C07276=1022.526,-49.278,404.640,166.557,49.308,158.966
C07277=1022.532,-49.029,404.628,166.560,49.304,158.966
C07278=1022.538,-48.778,404.616,166.563,49.300,158.966
C07279=1022.544,-48.529,404.605,166.566,49.296,158.965
C07280=1022.550,-48.279,404.592,166.568,49.292,158.965
C07281=1022.555,-48.030,404.581,166.572,49.289,158.965
C07282=1022.561,-47.780,404.569,166.574,49.285,158.965
C07283=1022.566,-47.530,404.557,166.577,49.281,158.964
C07284=1022.573,-47.281,404.545,166.580,49.277,158.964
C07285=1022.578,-47.031,404.534,166.583,49.274,158.964
C07286=1022.585,-46.781,404.522,166.586,49.270,158.964
C07287=1022.590,-46.532,404.510,166.588,49.266,158.963
C07288=1022.596,-46.282,404.498,166.592,49.263,158.963
C07289=1022.601,-46.033,404.486,166.594,49.259,158.963
C07290=1022.607,-45.783,404.474,166.598,49.254,158.963
C07291=1022.613,-45.533,404.463,166.601,49.251,158.963
C07292=1022.619,-45.284,404.450,166.604,49.247,158.962
C07293=1022.625,-45.035,404.439,166.607,49.243,158.962
C07294=1022.631,-44.784,404.427,166.610,49.239,158.962
C07295=1022.636,-44.535,404.415,166.613,49.236,158.962
C07296=1022.643,-44.285,404.403,166.615,49.232,158.961
C07297=1022.648,-44.035,404.391,166.618,49.228,158.961
C07298=1022.654,-43.786,404.379,166.621,49.224,158.961
C07299=1022.660,-43.536,404.367,166.624,49.221,158.961
C07300=1022.666,-43.287,404.356,166.627,49.217,158.960
C07301=1022.672,-43.037,404.343,166.630,49.213,158.960
C07302=1022.677,-42.788,404.331,166.632,49.209,158.960
C07303=1022.684,-42.538,404.319,166.635,49.205,158.960
C07304=1022.689,-42.288,404.307,166.638,49.201,158.959
C07305=1022.695,-42.039,404.296,166.642,49.197,158.959
C07306=1022.701,-41.789,404.283,166.645,49.193,158.959
C07307=1022.707,-41.539,404.271,166.648,49.189,158.958
C07308=1022.713,-41.289,404.260,166.651,49.186,158.958
C07309=1022.719,-41.040,404.247,166.653,49.182,158.958
C07310=1022.725,-40.791,404.236,166.656,49.178,158.958
C07311=1022.731,-40.541,404.223,166.659,49.174,158.957
C07312=1022.737,-40.291,404.210,166.662,49.170,158.957
C07313=1022.743,-40.041,404.200,166.665,49.167,158.957
C07314=1022.748,-39.792,404.187,166.668,49.163,158.957
C07315=1022.755,-39.542,404.175,166.670,49.159,158.956
C07316=1022.760,-39.293,404.163,166.673,49.155,158.956
C07317=1022.766,-39.043,404.150,166.676,49.151,158.956
C07318=1022.772,-38.793,404.138,166.679,49.147,158.956
C07319=1022.779,-38.543,404.126,166.682,49.143,158.955
C07320=1022.784,-38.294,404.114,166.685,49.139,158.955
C07321=1022.790,-38.044,404.101,166.688,49.136,158.955
C07322=1022.796,-37.794,404.089,166.690,49.132,158.955
C07323=1022.801,-37.545,404.077,166.693,49.128,158.954
C07324=1022.808,-37.266,404.063,166.697,49.124,158.954
C07325=1022.815,-36.986,404.049,166.700,49.120,158.954
C07326=1022.821,-36.708,404.035,166.704,49.116,158.954
C07327=1022.828,-36.429,404.021,166.706,49.112,158.953
C07328=1022.834,-36.179,404.008,166.709,49.108,158.953
C07329=1022.839,-35.929,403.996,166.712,49.104,158.953
C07330=1022.845,-35.680,403.984,166.715,49.100,158.953
C07331=1022.851,-35.430,403.972,166.718,49.096,158.952
C07332=1022.857,-35.180,403.959,166.721,49.093,158.952
C07333=1022.863,-34.931,403.947,166.724,49.089,158.952
C07334=1022.869,-34.681,403.934,166.726,49.085,158.952
C07335=1022.875,-34.431,403.922,166.729,49.081,158.951
C07336=1022.880,-34.181,403.909,166.732,49.078,158.951
C07337=1022.886,-33.932,403.897,166.735,49.074,158.951
C07338=1022.892,-33.682,403.885,166.738,49.070,158.951
C07339=1022.898,-33.433,403.873,166.741,49.066,158.950
C07340=1022.904,-33.183,403.859,166.744,49.063,158.950
C07341=1022.910,-32.934,403.847,166.747,49.059,158.950
C07342=1022.916,-32.684,403.835,166.749,49.055,158.950
C07343=1022.922,-32.434,403.822,166.752,49.051,158.949
C07344=1022.928,-32.185,403.809,166.755,49.048,158.949
C07345=1022.933,-31.935,403.797,166.758,49.044,158.949
C07346=1022.939,-31.686,403.785,166.761,49.040,158.949
C07347=1022.945,-31.436,403.771,166.764,49.036,158.948
C07348=1022.952,-31.187,403.760,166.767,49.032,158.948
C07349=1022.958,-30.937,403.747,166.769,49.028,158.948
C07350=1022.963,-30.687,403.734,166.772,49.024,158.948
C07351=1022.969,-30.437,403.722,166.775,49.020,158.947
C07352=1022.975,-30.188,403.709,166.778,49.017,158.947
C07353=1022.981,-29.939,403.696,166.781,49.013,158.947
C07354=1022.987,-29.689,403.684,166.784,49.009,158.946
C07355=1022.993,-29.439,403.671,166.786,49.005,158.946
C07356=1022.999,-29.189,403.659,166.789,49.001,158.946
C07357=1023.006,-28.940,403.646,166.792,48.997,158.946
C07358=1023.011,-28.690,403.634,166.795,48.994,158.945
C07359=1023.017,-28.441,403.621,166.798,48.990,158.945
C07360=1023.023,-28.192,403.608,166.801,48.986,158.945
C07361=1023.029,-27.942,403.595,166.804,48.982,158.945
C07362=1023.035,-27.692,403.583,166.807,48.978,158.944
C07363=1023.041,-27.442,403.570,166.810,48.974,158.944
C07364=1023.047,-27.193,403.557,166.812,48.971,158.944
C07365=1023.053,-26.943,403.545,166.815,48.967,158.943
C07366=1023.059,-26.694,403.531,166.818,48.963,158.943
C07367=1023.064,-26.443,403.518,166.821,48.960,158.943
C07368=1023.070,-26.194,403.506,166.824,48.956,158.943
C07369=1023.076,-25.945,403.493,166.826,48.952,158.942
C07370=1023.082,-25.695,403.480,166.829,48.949,158.942
C07371=1023.088,-25.446,403.467,166.832,48.945,158.942
C07372=1023.094,-25.196,403.454,166.835,48.941,158.942
C07373=1023.099,-24.946,403.440,166.838,48.938,158.942
C07374=1023.105,-24.696,403.428,166.841,48.934,158.941
C07375=1023.111,-24.447,403.415,166.844,48.930,158.941
C07376=1023.117,-24.197,403.402,166.847,48.926,158.941
C07377=1023.123,-23.948,403.389,166.850,48.922,158.941
C07378=1023.129,-23.698,403.376,166.852,48.918,158.940
C07379=1023.135,-23.449,403.362,166.854,48.915,158.940
C07380=1023.141,-23.199,403.350,166.857,48.912,158.940
C07381=1023.147,-22.949,403.337,166.860,48.908,158.939
C07382=1023.153,-22.700,403.324,166.863,48.904,158.939
C07383=1023.159,-22.450,403.311,166.866,48.900,158.939
C07384=1023.164,-22.200,403.298,166.869,48.896,158.939
C07385=1023.170,-21.951,403.284,166.871,48.892,158.938
C07386=1023.176,-21.701,403.272,166.874,48.889,158.938
C07387=1023.183,-21.452,403.258,166.877,48.885,158.938
C07388=1023.189,-21.172,403.244,166.880,48.881,158.937
C07389=1023.196,-20.892,403.229,166.884,48.876,158.937
C07390=1023.202,-20.612,403.214,166.886,48.872,158.937
C07391=1023.209,-20.332,403.200,166.890,48.867,158.937
C07392=1023.215,-20.083,403.187,166.893,48.864,158.936
C07393=1023.221,-19.833,403.174,166.896,48.860,158.936
C07394=1023.227,-19.582,403.160,166.899,48.856,158.936
C07395=1023.233,-19.333,403.147,166.901,48.852,158.935
C07396=1023.239,-19.084,403.134,166.903,48.849,158.935
C07397=1023.245,-18.834,403.121,166.906,48.845,158.935
C07398=1023.251,-18.585,403.108,166.909,48.842,158.935
C07399=1023.257,-18.335,403.094,166.912,48.838,158.934
C07400=1023.263,-18.085,403.081,166.915,48.834,158.934
C07401=1023.269,-17.836,403.068,166.917,48.830,158.934
C07402=1023.275,-17.587,403.055,166.921,48.826,158.934
C07403=1023.281,-17.337,403.042,166.923,48.822,158.933
C07404=1023.287,-17.087,403.028,166.926,48.819,158.933
C07405=1023.293,-16.838,403.015,166.929,48.815,158.933
C07406=1023.299,-16.588,403.003,166.932,48.811,158.932
C07407=1023.305,-16.339,402.989,166.934,48.807,158.932
C07408=1023.312,-16.089,402.976,166.938,48.803,158.932
C07409=1023.317,-15.839,402.962,166.940,48.800,158.932
C07410=1023.323,-15.589,402.949,166.943,48.796,158.931
C07411=1023.329,-15.340,402.936,166.946,48.792,158.931
C07412=1023.335,-15.091,402.922,166.949,48.788,158.931
C07413=1023.341,-14.841,402.909,166.951,48.785,158.930
C07414=1023.346,-14.592,402.895,166.954,48.781,158.930
C07415=1023.353,-14.343,402.882,166.956,48.777,158.930
C07416=1023.359,-14.092,402.868,166.960,48.774,158.930
C07417=1023.365,-13.842,402.855,166.962,48.770,158.929
C07418=1023.370,-13.593,402.841,166.965,48.766,158.929
C07419=1023.376,-13.344,402.828,166.968,48.763,158.929
C07420=1023.382,-13.094,402.814,166.971,48.759,158.929
C07421=1023.388,-12.845,402.801,166.973,48.755,158.928
C07422=1023.394,-12.595,402.787,166.976,48.751,158.928
C07423=1023.400,-12.345,402.773,166.979,48.748,158.928
C07424=1023.406,-12.096,402.759,166.982,48.744,158.927
C07425=1023.412,-11.846,402.746,166.984,48.740,158.927
C07426=1023.418,-11.597,402.732,166.987,48.736,158.927
C07427=1023.424,-11.347,402.719,166.990,48.733,158.927
C07428=1023.429,-11.098,402.705,166.993,48.729,158.926
C07429=1023.436,-10.848,402.691,166.996,48.725,158.926
C07430=1023.442,-10.598,402.678,166.998,48.721,158.926
C07431=1023.448,-10.349,402.664,167.001,48.718,158.925
C07432=1023.454,-10.100,402.651,167.004,48.714,158.925
C07433=1023.459,-9.850,402.637,167.006,48.710,158.925
C07434=1023.466,-9.600,402.624,167.009,48.706,158.924
C07435=1023.472,-9.351,402.610,167.012,48.703,158.924
C07436=1023.478,-9.101,402.596,167.015,48.699,158.924
C07437=1023.483,-8.852,402.583,167.018,48.695,158.924
C07438=1023.490,-8.602,402.569,167.021,48.691,158.923
C07439=1023.496,-8.352,402.555,167.022,48.687,158.923
C07440=1023.502,-8.103,402.542,167.025,48.684,158.923
C07441=1023.507,-7.854,402.528,167.028,48.680,158.923
C07442=1023.514,-7.604,402.515,167.031,48.676,158.922
C07443=1023.520,-7.354,402.500,167.034,48.672,158.922
C07444=1023.526,-7.105,402.487,167.037,48.669,158.922
C07445=1023.531,-6.855,402.473,167.039,48.665,158.921
C07446=1023.538,-6.605,402.460,167.042,48.661,158.921
C07447=1023.544,-6.356,402.445,167.045,48.657,158.921
C07448=1023.550,-6.107,402.432,167.047,48.654,158.920
C07449=1023.556,-5.857,402.418,167.050,48.650,158.920
C07450=1023.562,-5.607,402.404,167.053,48.646,158.920
C07451=1023.568,-5.358,402.390,167.056,48.642,158.919
C07452=1023.575,-5.076,402.375,167.059,48.638,158.919
C07453=1023.582,-4.794,402.359,167.062,48.633,158.919
C07454=1023.589,-4.513,402.344,167.065,48.629,158.918
C07455=1023.596,-4.231,402.329,167.069,48.625,158.918
C07456=1023.602,-3.981,402.314,167.071,48.621,158.918
C07457=1023.607,-3.732,402.300,167.073,48.618,158.917
C07458=1023.613,-3.483,402.286,167.076,48.614,158.917
C07459=1023.619,-3.232,402.272,167.079,48.610,158.917
C07460=1023.625,-2.983,402.258,167.082,48.606,158.917
C07461=1023.631,-2.734,402.244,167.085,48.603,158.917
C07462=1023.637,-2.484,402.230,167.087,48.600,158.916
C07463=1023.643,-2.234,402.216,167.090,48.596,158.916
C07464=1023.648,-1.985,402.201,167.093,48.592,158.916
C07465=1023.654,-1.735,402.187,167.095,48.589,158.915
C07466=1023.660,-1.486,402.172,167.098,48.585,158.915
C07467=1023.666,-1.236,402.158,167.100,48.582,158.915
C07468=1023.672,-0.986,402.144,167.103,48.578,158.915
C07469=1023.678,-0.738,402.130,167.106,48.574,158.914
C07470=1023.684,-0.488,402.116,167.109,48.570,158.914
C07471=1023.690,-0.238,402.101,167.112,48.567,158.914
C07472=1023.696,0.011,402.088,167.114,48.563,158.913
C07473=1023.701,0.261,402.074,167.116,48.559,158.913
C07474=1023.707,0.510,402.059,167.120,48.556,158.913
C07475=1023.713,0.760,402.045,167.122,48.552,158.913
C07476=1023.719,1.009,402.031,167.125,48.548,158.912
C07477=1023.726,1.259,402.017,167.127,48.545,158.912
C07478=1023.731,1.508,402.002,167.130,48.541,158.912
C07479=1023.737,1.758,401.988,167.133,48.537,158.911
C07480=1023.743,2.007,401.973,167.136,48.533,158.911
C07481=1023.749,2.257,401.959,167.139,48.530,158.911
C07482=1023.755,2.507,401.945,167.141,48.527,158.910
C07483=1023.761,2.756,401.931,167.143,48.523,158.910
C07484=1023.767,3.006,401.917,167.146,48.519,158.910
C07485=1023.773,3.255,401.902,167.149,48.515,158.909
C07486=1023.779,3.504,401.888,167.152,48.512,158.909
C07487=1023.785,3.754,401.874,167.154,48.508,158.909
C07488=1023.791,4.003,401.859,167.157,48.504,158.909
C07489=1023.797,4.253,401.845,167.160,48.500,158.908
C07490=1023.803,4.502,401.830,167.162,48.496,158.908
C07491=1023.809,4.753,401.816,167.166,48.493,158.908
C07492=1023.814,5.002,401.801,167.167,48.489,158.907
C07493=1023.821,5.251,401.788,167.170,48.486,158.907
C07494=1023.827,5.500,401.773,167.173,48.482,158.907
C07495=1023.833,5.751,401.759,167.176,48.478,158.906
C07496=1023.839,6.000,401.744,167.179,48.474,158.906
C07497=1023.845,6.249,401.729,167.182,48.471,158.906
C07498=1023.851,6.499,401.716,167.183,48.467,158.906
C07499=1023.857,6.749,401.701,167.186,48.463,158.905
C07500=1023.863,6.998,401.687,167.189,48.459,158.905
C07501=1023.869,7.248,401.672,167.192,48.455,158.905
C07502=1023.876,7.496,401.658,167.195,48.451,158.904
C07503=1023.882,7.747,401.644,167.197,48.449,158.904
C07504=1023.887,7.996,401.629,167.200,48.445,158.904
C07505=1023.894,8.245,401.614,167.202,48.441,158.903
C07506=1023.899,8.495,401.600,167.205,48.437,158.903
C07507=1023.906,8.745,401.585,167.208,48.433,158.903
C07508=1023.911,8.994,401.571,167.211,48.429,158.902
C07509=1023.918,9.244,401.556,167.213,48.425,158.902
C07510=1023.923,9.493,401.542,167.215,48.421,158.902
C07511=1023.930,9.742,401.527,167.218,48.418,158.901
C07512=1023.936,9.992,401.514,167.221,48.414,158.901
C07513=1023.942,10.241,401.499,167.224,48.410,158.901
C07514=1023.948,10.490,401.484,167.227,48.407,158.901
C07515=1023.954,10.740,401.469,167.229,48.403,158.900
C07516=1023.962,11.023,401.453,167.232,48.398,158.900
C07517=1023.968,11.307,401.436,167.235,48.394,158.899
C07518=1023.975,11.591,401.419,167.238,48.390,158.899
C07519=1023.982,11.874,401.403,167.242,48.385,158.899
C07520=1023.988,12.124,401.389,167.244,48.382,158.898
C07521=1023.994,12.373,401.374,167.247,48.378,158.898
C07522=1024.000,12.623,401.359,167.249,48.374,158.898
C07523=1024.007,12.873,401.344,167.252,48.370,158.897
C07524=1024.012,13.122,401.330,167.255,48.366,158.897
C07525=1024.019,13.372,401.316,167.257,48.362,158.897
C07526=1024.025,13.622,401.301,167.260,48.358,158.896
C07527=1024.031,13.871,401.286,167.262,48.356,158.896
C07528=1024.037,14.120,401.271,167.265,48.352,158.896
C07529=1024.043,14.369,401.257,167.268,48.348,158.895
C07530=1024.049,14.619,401.242,167.271,48.344,158.895
C07531=1024.055,14.869,401.226,167.273,48.340,158.895
C07532=1024.061,15.118,401.211,167.276,48.337,158.895
C07533=1024.067,15.367,401.197,167.278,48.333,158.894
C07534=1024.073,15.616,401.182,167.281,48.329,158.894
C07535=1024.079,15.866,401.167,167.284,48.325,158.894
C07536=1024.085,16.117,401.152,167.286,48.322,158.893
C07537=1024.090,16.366,401.138,167.289,48.319,158.893
C07538=1024.097,16.615,401.123,167.292,48.315,158.893
C07539=1024.103,16.865,401.108,167.295,48.311,158.892
C07540=1024.109,17.114,401.093,167.296,48.307,158.892
C07541=1024.115,17.364,401.078,167.299,48.303,158.892
C07542=1024.121,17.613,401.063,167.302,48.299,158.891
C07543=1024.127,17.862,401.048,167.305,48.296,158.891
C07544=1024.133,18.112,401.033,167.307,48.293,158.891
C07545=1024.139,18.362,401.018,167.310,48.289,158.890
C07546=1024.145,18.610,401.002,167.313,48.285,158.890
C07547=1024.151,18.860,400.987,167.316,48.281,158.890
C07548=1024.158,19.110,400.972,167.317,48.277,158.889
C07549=1024.163,19.359,400.958,167.320,48.274,158.889
C07550=1024.169,19.609,400.942,167.323,48.270,158.889
C07551=1024.175,19.858,400.927,167.326,48.266,158.888
C07552=1024.182,20.108,400.912,167.328,48.263,158.888
C07553=1024.187,20.357,400.897,167.331,48.259,158.888
C07554=1024.193,20.607,400.882,167.334,48.255,158.887
C07555=1024.200,20.857,400.867,167.336,48.251,158.887
C07556=1024.205,21.105,400.851,167.339,48.248,158.887
C07557=1024.211,21.355,400.836,167.341,48.244,158.886
C07558=1024.218,21.604,400.822,167.344,48.241,158.886
C07559=1024.223,21.854,400.806,167.347,48.237,158.886
C07560=1024.229,22.103,400.791,167.349,48.233,158.885
C07561=1024.235,22.353,400.776,167.352,48.229,158.885
C07562=1024.241,22.602,400.760,167.355,48.226,158.885
C07563=1024.247,22.851,400.746,167.358,48.222,158.885
C07564=1024.254,23.101,400.731,167.359,48.219,158.884
C07565=1024.259,23.351,400.715,167.362,48.215,158.884
C07566=1024.266,23.601,400.700,167.365,48.211,158.884
C07567=1024.272,23.850,400.684,167.368,48.207,158.883
C07568=1024.277,24.099,400.669,167.370,48.203,158.883
C07569=1024.284,24.349,400.654,167.373,48.200,158.883
C07570=1024.289,24.599,400.639,167.376,48.196,158.882
C07571=1024.296,24.848,400.623,167.378,48.192,158.882
C07572=1024.302,25.097,400.609,167.380,48.189,158.882
C07573=1024.308,25.347,400.593,167.383,48.185,158.881
C07574=1024.314,25.596,400.578,167.386,48.181,158.881
C07575=1024.321,25.845,400.562,167.389,48.177,158.881
C07576=1024.326,26.095,400.547,167.391,48.174,158.880
C07577=1024.332,26.344,400.532,167.394,48.170,158.880
C07578=1024.338,26.593,400.516,167.397,48.167,158.880
C07579=1024.344,26.843,400.501,167.398,48.163,158.879
C07580=1024.351,27.128,400.483,167.402,48.158,158.879
C07581=1024.358,27.413,400.466,167.405,48.154,158.878
C07582=1024.365,27.698,400.448,167.407,48.150,158.878
C07583=1024.372,27.983,400.430,167.411,48.146,158.878
C07584=1024.378,28.233,400.415,167.413,48.142,158.877
C07585=1024.384,28.482,400.399,167.416,48.138,158.877
C07586=1024.390,28.731,400.384,167.419,48.135,158.877
C07587=1024.396,28.981,400.369,167.421,48.131,158.876
C07588=1024.402,29.230,400.352,167.423,48.127,158.876
C07589=1024.408,29.480,400.337,167.426,48.124,158.876
C07590=1024.414,29.729,400.321,167.428,48.120,158.875
C07591=1024.420,29.978,400.307,167.431,48.117,158.875
C07592=1024.426,30.228,400.290,167.434,48.113,158.875
C07593=1024.431,30.478,400.275,167.436,48.109,158.874
C07594=1024.438,30.727,400.259,167.439,48.106,158.874
C07595=1024.444,30.977,400.244,167.442,48.102,158.874
C07596=1024.450,31.226,400.228,167.444,48.098,158.873
C07597=1024.456,31.476,400.212,167.447,48.095,158.873
C07598=1024.461,31.724,400.197,167.449,48.091,158.873
C07599=1024.468,31.974,400.182,167.452,48.087,158.872
C07600=1024.474,32.223,400.165,167.454,48.084,158.872
C07601=1024.480,32.473,400.150,167.457,48.080,158.872
C07602=1024.486,32.722,400.134,167.460,48.076,158.871
C07603=1024.492,32.972,400.118,167.462,48.072,158.871
C07604=1024.498,33.221,400.103,167.465,48.069,158.871
C07605=1024.504,33.471,400.087,167.467,48.065,158.870
C07606=1024.510,33.721,400.071,167.470,48.061,158.870
C07607=1024.516,33.969,400.056,167.472,48.058,158.870
C07608=1024.522,34.219,400.040,167.475,48.054,158.869
C07609=1024.528,34.468,400.025,167.478,48.050,158.869
C07610=1024.534,34.717,400.008,167.481,48.046,158.869
C07611=1024.540,34.967,399.993,167.482,48.043,158.868
C07612=1024.547,35.216,399.977,167.485,48.039,158.868
C07613=1024.552,35.466,399.962,167.488,48.035,158.868
C07614=1024.558,35.716,399.945,167.490,48.032,158.867
C07615=1024.565,35.965,399.930,167.493,48.028,158.867
C07616=1024.570,36.215,399.914,167.496,48.024,158.867
C07617=1024.577,36.464,399.899,167.499,48.021,158.866
C07618=1024.583,36.713,399.882,167.501,48.017,158.866
C07619=1024.589,36.963,399.867,167.503,48.013,158.866
C07620=1024.595,37.212,399.850,167.506,48.009,158.865
C07621=1024.601,37.462,399.834,167.508,48.006,158.865
C07622=1024.607,37.711,399.819,167.511,48.002,158.865
C07623=1024.613,37.961,399.803,167.514,47.999,158.864
C07624=1024.619,38.210,399.787,167.516,47.995,158.864
C07625=1024.625,38.460,399.770,167.519,47.991,158.864
C07626=1024.631,38.709,399.754,167.522,47.987,158.863
C07627=1024.637,38.958,399.738,167.523,47.984,158.863
C07628=1024.642,39.208,399.722,167.526,47.981,158.863
C07629=1024.649,39.457,399.707,167.529,47.977,158.862
C07630=1024.655,39.706,399.691,167.531,47.973,158.862
C07631=1024.660,39.955,399.675,167.534,47.969,158.862
C07632=1024.666,40.205,399.658,167.537,47.966,158.861
C07633=1024.672,40.454,399.642,167.539,47.962,158.861
C07634=1024.678,40.704,399.627,167.542,47.959,158.861
C07635=1024.685,40.954,399.610,167.545,47.955,158.860
C07636=1024.691,41.203,399.594,167.546,47.951,158.860
C07637=1024.697,41.452,399.578,167.549,47.948,158.860
C07638=1024.703,41.702,399.562,167.552,47.944,158.859
C07639=1024.709,41.951,399.546,167.554,47.940,158.859
C07640=1024.715,42.200,399.529,167.557,47.936,158.858
C07641=1024.721,42.450,399.513,167.560,47.932,158.858
C07642=1024.727,42.700,399.497,167.562,47.930,158.858
C07643=1024.733,42.949,399.481,167.565,47.926,158.857
C07644=1024.739,43.233,399.463,167.567,47.922,158.857
C07645=1024.746,43.518,399.444,167.570,47.917,158.857
C07646=1024.753,43.804,399.425,167.573,47.913,158.856
C07647=1024.759,44.089,399.406,167.577,47.909,158.856
C07648=1024.765,44.338,399.389,167.579,47.906,158.856
C07649=1024.771,44.588,399.373,167.581,47.902,158.855
C07650=1024.777,44.837,399.357,167.584,47.899,158.855
C07651=1024.783,45.086,399.341,167.586,47.895,158.855
C07652=1024.789,45.336,399.324,167.589,47.891,158.854
C07653=1024.795,45.585,399.308,167.591,47.888,158.854
C07654=1024.800,45.835,399.291,167.594,47.885,158.854
C07655=1024.806,46.084,399.275,167.596,47.881,158.853
C07656=1024.812,46.333,399.258,167.599,47.877,158.853
C07657=1024.818,46.582,399.242,167.602,47.873,158.853
C07658=1024.824,46.831,399.226,167.604,47.871,158.852
C07659=1024.830,47.081,399.209,167.607,47.867,158.852
C07660=1024.836,47.330,399.192,167.610,47.863,158.852
C07661=1024.842,47.580,399.176,167.611,47.859,158.851
C07662=1024.848,47.830,399.160,167.614,47.856,158.851
C07663=1024.854,48.079,399.143,167.616,47.853,158.851
C07664=1024.860,48.328,399.126,167.619,47.849,158.850
C07665=1024.866,48.577,399.110,167.622,47.845,158.850
C07666=1024.871,48.827,399.093,167.624,47.841,158.850
C07667=1024.877,49.076,399.077,167.627,47.838,158.849
C07668=1024.883,49.326,399.061,167.630,47.834,158.849
C07669=1024.889,49.575,399.045,167.632,47.831,158.849
C07670=1024.896,49.824,399.028,167.635,47.827,158.848
C07671=1024.902,50.074,399.011,167.637,47.823,158.848
C07672=1024.907,50.323,398.994,167.639,47.820,158.848
C07673=1024.913,50.573,398.978,167.642,47.816,158.847
C07674=1024.919,50.822,398.962,167.645,47.813,158.847
C07675=1024.925,51.071,398.945,167.647,47.809,158.847
C07676=1024.931,51.320,398.928,167.650,47.805,158.846
C07677=1024.938,51.570,398.912,167.652,47.802,158.846
C07678=1024.943,51.820,398.895,167.655,47.798,158.845
C07679=1024.949,52.069,398.878,167.657,47.794,158.845
C07680=1024.955,52.318,398.862,167.659,47.791,158.845
C07681=1024.961,52.567,398.845,167.662,47.787,158.844
C07682=1024.967,52.817,398.829,167.665,47.784,158.844
C07683=1024.973,53.066,398.811,167.667,47.780,158.844
C07684=1024.979,53.316,398.795,167.670,47.776,158.843
C07685=1024.985,53.565,398.779,167.673,47.772,158.843
C07686=1024.991,53.814,398.762,167.675,47.769,158.843
C07687=1024.998,54.063,398.745,167.678,47.765,158.842
C07688=1025.004,54.313,398.729,167.680,47.761,158.842
C07689=1025.009,54.563,398.712,167.682,47.758,158.842
C07690=1025.016,54.812,398.695,167.685,47.754,158.841
C07691=1025.021,55.061,398.679,167.688,47.750,158.841
C07692=1025.028,55.311,398.662,167.690,47.747,158.841
C07693=1025.034,55.560,398.645,167.693,47.743,158.840
C07694=1025.040,55.809,398.628,167.696,47.739,158.840
C07695=1025.045,56.059,398.612,167.698,47.736,158.840
C07696=1025.052,56.308,398.595,167.700,47.732,158.839
C07697=1025.058,56.558,398.578,167.703,47.728,158.839
C07698=1025.064,56.807,398.562,167.705,47.725,158.838
C07699=1025.070,57.056,398.545,167.708,47.721,158.838
C07700=1025.076,57.306,398.528,167.711,47.717,158.838
C07701=1025.083,57.555,398.511,167.714,47.713,158.837
C07702=1025.089,57.804,398.495,167.716,47.710,158.837
C07703=1025.094,58.053,398.479,167.718,47.706,158.837
C07704=1025.101,58.303,398.461,167.721,47.702,158.836
C07705=1025.107,58.552,398.444,167.723,47.699,158.836
C07706=1025.113,58.801,398.427,167.726,47.695,158.835
C07707=1025.119,59.051,398.411,167.729,47.691,158.835
C07708=1025.126,59.335,398.392,167.732,47.687,158.835
C07709=1025.133,59.620,398.372,167.734,47.683,158.834
C07710=1025.140,59.905,398.353,167.737,47.678,158.834
C07711=1025.147,60.190,398.334,167.741,47.674,158.833
C07712=1025.153,60.439,398.317,167.743,47.671,158.833
C07713=1025.160,60.689,398.300,167.745,47.667,158.833
C07714=1025.165,60.938,398.284,167.748,47.663,158.832
C07715=1025.171,61.187,398.266,167.750,47.659,158.832
C07716=1025.178,61.437,398.250,167.753,47.656,158.832
C07717=1025.184,61.686,398.233,167.756,47.652,158.831
C07718=1025.190,61.935,398.217,167.758,47.648,158.831
C07719=1025.197,62.185,398.199,167.761,47.644,158.830
C07720=1025.202,62.434,398.182,167.763,47.641,158.830
C07721=1025.208,62.683,398.165,167.766,47.637,158.830
C07722=1025.215,62.933,398.149,167.768,47.633,158.829
C07723=1025.221,63.182,398.132,167.771,47.629,158.829
C07724=1025.227,63.431,398.114,167.774,47.626,158.829
C07725=1025.233,63.681,398.098,167.776,47.622,158.828
C07726=1025.238,63.930,398.080,167.778,47.618,158.828
C07727=1025.245,64.180,398.063,167.781,47.614,158.828
C07728=1025.251,64.429,398.046,167.783,47.611,158.827
C07729=1025.257,64.678,398.029,167.786,47.607,158.827
C07730=1025.263,64.928,398.012,167.789,47.603,158.826
C07731=1025.269,65.177,397.995,167.791,47.600,158.826
C07732=1025.278,65.553,397.968,167.795,47.594,158.825
C07733=1025.287,65.929,397.943,167.799,47.589,158.825
C07734=1025.296,66.305,397.916,167.803,47.584,158.824
C07735=1025.305,66.680,397.891,167.806,47.578,158.824
C07736=1025.310,66.929,397.873,167.809,47.574,158.824
C07737=1025.317,67.179,397.856,167.811,47.571,158.823
C07738=1025.323,67.428,397.838,167.814,47.567,158.823
C07739=1025.329,67.678,397.822,167.817,47.563,158.822
C07740=1025.335,67.927,397.804,167.819,47.560,158.822
C07741=1025.340,68.176,397.786,167.821,47.556,158.822
C07742=1025.347,68.426,397.769,167.825,47.553,158.821
C07743=1025.353,68.675,397.752,167.826,47.549,158.821
C07744=1025.359,68.925,397.735,167.829,47.545,158.821
C07745=1025.365,69.174,397.717,167.832,47.542,158.820
C07746=1025.370,69.423,397.700,167.834,47.538,158.820
C07747=1025.377,69.672,397.682,167.837,47.534,158.820
C07748=1025.383,69.921,397.665,167.839,47.531,158.819
C07749=1025.389,70.171,397.647,167.842,47.528,158.819
C07750=1025.394,70.420,397.629,167.845,47.524,158.819
C07751=1025.401,70.669,397.612,167.847,47.520,158.818
C07752=1025.406,70.919,397.595,167.849,47.517,158.818
C07753=1025.412,71.168,397.578,167.852,47.513,158.817
C07754=1025.419,71.417,397.560,167.854,47.509,158.817
C07755=1025.424,71.667,397.543,167.857,47.506,158.817
C07756=1025.431,71.916,397.525,167.860,47.502,158.816
C07757=1025.436,72.165,397.507,167.862,47.499,158.816
C07758=1025.443,72.415,397.490,167.865,47.495,158.816
C07759=1025.448,72.664,397.472,167.867,47.492,158.815
C07760=1025.455,72.914,397.454,167.870,47.488,158.815
C07761=1025.460,73.163,397.437,167.873,47.484,158.815
C07762=1025.467,73.412,397.419,167.874,47.480,158.814
C07763=1025.472,73.661,397.402,167.877,47.477,158.814
C07764=1025.479,73.911,397.384,167.880,47.473,158.813
C07765=1025.484,74.160,397.366,167.882,47.469,158.813
C07766=1025.491,74.409,397.349,167.885,47.466,158.813
C07767=1025.496,74.658,397.331,167.888,47.462,158.812
C07768=1025.506,75.066,397.303,167.892,47.456,158.812
C07769=1025.516,75.473,397.274,167.895,47.451,158.811
C07770=1025.525,75.880,397.245,167.899,47.444,158.810
C07771=1025.536,76.288,397.216,167.904,47.439,158.810
C07772=1025.541,76.537,397.199,167.907,47.435,158.810
C07773=1025.548,76.787,397.181,167.909,47.431,158.809
C07774=1025.553,77.035,397.162,167.911,47.428,158.809
C07775=1025.560,77.285,397.144,167.914,47.424,158.809
C07776=1025.565,77.534,397.127,167.917,47.421,158.808
C07777=1025.572,77.784,397.110,167.919,47.417,158.808
C07778=1025.577,78.033,397.092,167.922,47.413,158.807
C07779=1025.583,78.283,397.073,167.924,47.410,158.807
C07780=1025.588,78.532,397.056,167.927,47.406,158.807
C07781=1025.595,78.781,397.037,167.930,47.403,158.807
C07782=1025.601,79.031,397.019,167.932,47.399,158.806
C07783=1025.606,79.280,397.002,167.935,47.396,158.806
C07784=1025.613,79.529,396.984,167.937,47.392,158.805
C07785=1025.618,79.778,396.965,167.939,47.388,158.805
C07786=1025.624,80.027,396.948,167.943,47.385,158.805
C07787=1025.630,80.276,396.930,167.945,47.382,158.804
C07788=1025.636,80.526,396.912,167.947,47.378,158.804
C07789=1025.642,80.775,396.894,167.949,47.374,158.804
C07790=1025.648,81.024,396.876,167.952,47.371,158.803
C07791=1025.654,81.274,396.858,167.955,47.367,158.803
C07792=1025.660,81.523,396.840,167.957,47.364,158.803
C07793=1025.666,81.772,396.822,167.960,47.360,158.802
C07794=1025.672,82.021,396.804,167.963,47.357,158.802
C07795=1025.678,82.270,396.785,167.965,47.353,158.801
C07796=1025.684,82.520,396.768,167.968,47.349,158.801
C07797=1025.690,82.769,396.750,167.970,47.346,158.801
C07798=1025.696,83.019,396.732,167.973,47.343,158.800
C07799=1025.702,83.267,396.714,167.976,47.339,158.800
C07800=1025.708,83.517,396.696,167.977,47.335,158.800
C07801=1025.714,83.766,396.677,167.980,47.332,158.799
C07802=1025.720,84.015,396.660,167.983,47.328,158.799
C07803=1025.726,84.265,396.642,167.985,47.324,158.799
C07804=1025.731,84.514,396.623,167.988,47.321,158.798
C07805=1025.737,84.764,396.605,167.991,47.317,158.798
C07806=1025.743,85.013,396.587,167.993,47.313,158.797
C07807=1025.749,85.262,396.569,167.996,47.310,158.797
C07808=1025.755,85.511,396.551,167.999,47.306,158.797
C07809=1025.762,85.761,396.532,168.001,47.303,158.796
C07810=1025.767,86.010,396.514,168.004,47.299,158.796
C07811=1025.773,86.259,396.497,168.006,47.295,158.796
C07812=1025.780,86.508,396.478,168.008,47.292,158.795
C07813=1025.785,86.757,396.460,168.011,47.288,158.795
C07814=1025.792,87.007,396.442,168.014,47.284,158.795
C07815=1025.798,87.256,396.424,168.016,47.281,158.794
C07816=1025.803,87.505,396.405,168.019,47.277,158.794
C07817=1025.810,87.755,396.388,168.022,47.273,158.793
C07818=1025.816,88.004,396.370,168.024,47.271,158.793
C07819=1025.822,88.253,396.351,168.027,47.267,158.793
C07820=1025.828,88.502,396.333,168.030,47.263,158.792
C07821=1025.833,88.752,396.314,168.032,47.259,158.792
C07822=1025.839,89.002,396.296,168.034,47.256,158.792
C07823=1025.845,89.250,396.278,168.037,47.252,158.791
C07824=1025.851,89.500,396.260,168.039,47.248,158.791
C07825=1025.858,89.749,396.241,168.042,47.245,158.790
C07826=1025.864,89.998,396.222,168.045,47.241,158.790
C07827=1025.869,90.247,396.205,168.047,47.238,158.790
C07828=1025.875,90.496,396.186,168.050,47.234,158.789
C07829=1025.881,90.747,396.167,168.052,47.231,158.789
C07830=1025.887,90.995,396.149,168.055,47.227,158.789
C07831=1025.893,91.244,396.130,168.058,47.223,158.788
C07832=1025.899,91.529,396.110,168.061,47.220,158.788
C07833=1025.907,91.814,396.088,168.063,47.216,158.788
C07834=1025.913,92.098,396.067,168.066,47.211,158.787
C07835=1025.920,92.382,396.046,168.069,47.208,158.787
C07836=1025.926,92.632,396.028,168.072,47.204,158.786
C07837=1025.932,92.881,396.008,168.074,47.200,158.786
C07838=1025.937,93.129,395.990,168.077,47.197,158.786
C07839=1025.943,93.380,395.972,168.080,47.194,158.785
C07840=1025.949,93.629,395.953,168.082,47.190,158.785
C07841=1025.956,93.878,395.934,168.085,47.186,158.785
C07842=1025.961,94.126,395.915,168.087,47.183,158.784
C07843=1025.967,94.376,395.897,168.089,47.179,158.784
C07844=1025.973,94.625,395.879,168.092,47.176,158.784
C07845=1025.979,94.875,395.860,168.095,47.172,158.783
C07846=1025.985,95.123,395.841,168.097,47.169,158.783
C07847=1025.991,95.373,395.823,168.100,47.165,158.782
C07848=1025.997,95.622,395.804,168.103,47.161,158.782
C07849=1026.003,95.872,395.785,168.105,47.158,158.782
C07850=1026.009,96.121,395.766,168.108,47.154,158.781
C07851=1026.014,96.370,395.749,168.111,47.151,158.781
C07852=1026.021,96.619,395.730,168.113,47.147,158.781
C07853=1026.026,96.869,395.711,168.116,47.144,158.780
C07854=1026.033,97.118,395.692,168.119,47.140,158.780
C07855=1026.039,97.367,395.673,168.121,47.136,158.779
C07856=1026.044,97.616,395.655,168.123,47.133,158.779
C07857=1026.050,97.865,395.637,168.126,47.129,158.779
C07858=1026.056,98.115,395.617,168.128,47.125,158.778
C07859=1026.063,98.364,395.599,168.131,47.122,158.778
C07860=1026.069,98.613,395.580,168.134,47.119,158.778
C07861=1026.075,98.862,395.561,168.136,47.115,158.777
C07862=1026.081,99.111,395.543,168.139,47.111,158.777
C07863=1026.086,99.361,395.524,168.142,47.108,158.777
C07864=1026.092,99.610,395.505,168.144,47.104,158.776
C07865=1026.098,99.859,395.486,168.147,47.100,158.776
C07866=1026.104,100.109,395.468,168.150,47.097,158.776
C07867=1026.110,100.358,395.448,168.152,47.094,158.775
C07868=1026.116,100.607,395.429,168.155,47.090,158.775
C07869=1026.122,100.856,395.411,168.158,47.086,158.774
C07870=1026.127,101.105,395.391,168.160,47.084,158.774
C07871=1026.133,101.355,395.372,168.163,47.080,158.774
C07872=1026.139,101.604,395.354,168.165,47.076,158.773
C07873=1026.145,101.853,395.334,168.167,47.073,158.773
C07874=1026.151,102.103,395.315,168.170,47.069,158.773
C07875=1026.157,102.352,395.296,168.173,47.066,158.772
C07876=1026.162,102.601,395.278,168.175,47.062,158.772
C07877=1026.168,102.850,395.258,168.178,47.059,158.772
C07878=1026.175,103.098,395.239,168.180,47.055,158.771
C07879=1026.180,103.348,395.220,168.183,47.052,158.771
C07880=1026.186,103.597,395.200,168.186,47.048,158.771
C07881=1026.193,103.846,395.182,168.188,47.045,158.770
C07882=1026.198,104.096,395.163,168.191,47.041,158.770
C07883=1026.204,104.345,395.143,168.194,47.037,158.770
C07884=1026.210,104.594,395.125,168.196,47.035,158.769
C07885=1026.216,104.844,395.105,168.199,47.031,158.769
C07886=1026.221,105.093,395.087,168.202,47.027,158.769
C07887=1026.228,105.342,395.068,168.204,47.024,158.768
C07888=1026.234,105.591,395.048,168.207,47.020,158.768
C07889=1026.239,105.840,395.029,168.210,47.017,158.768
C07890=1026.246,106.089,395.010,168.212,47.013,158.767
C07891=1026.251,106.339,394.991,168.215,47.010,158.767
C07892=1026.257,106.588,394.972,168.218,47.006,158.766
C07893=1026.263,106.837,394.953,168.220,47.002,158.766
C07894=1026.269,107.086,394.933,168.222,46.999,158.766
C07895=1026.275,107.335,394.914,168.226,46.996,158.765
C07896=1026.281,107.620,394.892,168.228,46.991,158.765
C07897=1026.288,107.905,394.870,168.231,46.988,158.764
C07898=1026.296,108.189,394.849,168.234,46.983,158.764
C07899=1026.302,108.473,394.826,168.238,46.979,158.764
C07900=1026.308,108.722,394.807,168.240,46.976,158.763
C07901=1026.314,108.972,394.788,168.243,46.972,158.763
C07902=1026.320,109.221,394.769,168.246,46.969,158.763
C07903=1026.326,109.470,394.749,168.249,46.965,158.762
C07904=1026.332,109.719,394.730,168.250,46.962,158.762
C07905=1026.338,109.968,394.711,168.253,46.958,158.761
C07906=1026.344,110.218,394.692,168.256,46.954,158.761
C07907=1026.350,110.467,394.672,168.258,46.951,158.761
C07908=1026.356,110.716,394.653,168.261,46.948,158.760
C07909=1026.361,110.965,394.634,168.264,46.944,158.760
C07910=1026.367,111.214,394.614,168.266,46.941,158.760
C07911=1026.373,111.464,394.595,168.269,46.937,158.759
C07912=1026.380,111.712,394.575,168.272,46.934,158.759
C07913=1026.385,111.962,394.556,168.274,46.930,158.759
C07914=1026.391,112.211,394.537,168.277,46.927,158.758
C07915=1026.397,112.460,394.517,168.280,46.923,158.758
C07916=1026.403,112.709,394.498,168.283,46.919,158.758
C07917=1026.409,112.958,394.478,168.285,46.916,158.757
C07918=1026.414,113.207,394.458,168.288,46.913,158.757
C07919=1026.421,113.458,394.439,168.290,46.910,158.757
C07920=1026.426,113.707,394.418,168.293,46.906,158.756
C07921=1026.432,113.956,394.398,168.296,46.902,158.756
C07922=1026.438,114.205,394.379,168.298,46.900,158.756
C07923=1026.444,114.454,394.359,168.301,46.896,158.755
C07924=1026.449,114.703,394.340,168.304,46.892,158.755
C07925=1026.455,114.952,394.320,168.306,46.889,158.755
C07926=1026.461,115.201,394.301,168.309,46.886,158.754
C07927=1026.466,115.451,394.280,168.312,46.882,158.754
C07928=1026.472,115.700,394.261,168.314,46.879,158.754
C07929=1026.478,115.949,394.241,168.317,46.875,158.753
C07930=1026.484,116.198,394.221,168.320,46.872,158.753
C07931=1026.490,116.447,394.202,168.322,46.869,158.753
C07932=1026.496,116.696,394.182,168.325,46.865,158.752
C07933=1026.501,116.945,394.162,168.328,46.862,158.752
C07934=1026.507,117.194,394.142,168.330,46.859,158.752
C07935=1026.513,117.443,394.122,168.333,46.855,158.751
C07936=1026.518,117.693,394.103,168.336,46.851,158.751
C07937=1026.524,117.942,394.083,168.338,46.849,158.751
C07938=1026.530,118.190,394.063,168.341,46.845,158.750
C07939=1026.536,118.440,394.043,168.344,46.841,158.750
C07940=1026.542,118.690,394.023,168.346,46.838,158.750
C07941=1026.548,118.938,394.003,168.349,46.835,158.749
C07942=1026.554,119.188,393.983,168.352,46.831,158.749
C07943=1026.560,119.437,393.963,168.355,46.828,158.749
C07944=1026.566,119.685,393.943,168.357,46.824,158.748
C07945=1026.571,119.935,393.924,168.360,46.821,158.748
C07946=1026.576,120.184,393.904,168.363,46.817,158.747
C07947=1026.582,120.433,393.884,168.365,46.814,158.747
C07948=1026.588,120.682,393.864,168.368,46.811,158.747
C07949=1026.595,120.932,393.844,168.371,46.807,158.746
C07950=1026.601,121.181,393.824,168.374,46.804,158.746
C07951=1026.607,121.429,393.804,168.376,46.800,158.746
C07952=1026.612,121.679,393.784,168.379,46.797,158.745
C07953=1026.618,121.928,393.764,168.382,46.794,158.745
C07954=1026.624,122.177,393.744,168.384,46.790,158.745
C07955=1026.630,122.426,393.724,168.387,46.786,158.744
C07956=1026.636,122.676,393.705,168.390,46.783,158.744
C07957=1026.641,122.925,393.684,168.393,46.780,158.744
C07958=1026.647,123.174,393.664,168.395,46.776,158.743
C07959=1026.653,123.422,393.644,168.398,46.773,158.743
C07960=1026.660,123.707,393.622,168.401,46.769,158.743
C07961=1026.667,123.992,393.598,168.405,46.765,158.742
C07962=1026.674,124.276,393.576,168.408,46.761,158.742
C07963=1026.681,124.560,393.553,168.411,46.757,158.741
C07964=1026.686,124.810,393.533,168.413,46.753,158.741
C07965=1026.692,125.059,393.513,168.417,46.750,158.741
C07966=1026.698,125.308,393.493,168.420,46.746,158.740
C07967=1026.705,125.557,393.473,168.421,46.743,158.740
C07968=1026.711,125.806,393.453,168.424,46.739,158.740
C07969=1026.716,126.055,393.432,168.428,46.736,158.739
C07970=1026.722,126.304,393.412,168.431,46.733,158.739
C07971=1026.728,126.553,393.393,168.432,46.729,158.739
C07972=1026.734,126.803,393.373,168.435,46.725,158.738
C07973=1026.740,127.052,393.353,168.439,46.722,158.738
C07974=1026.745,127.301,393.332,168.441,46.719,158.738
C07975=1026.752,127.550,393.312,168.444,46.715,158.737
C07976=1026.758,127.799,393.292,168.446,46.712,158.737
C07977=1026.764,128.048,393.272,168.450,46.709,158.737
C07978=1026.770,128.297,393.252,168.452,46.705,158.736
C07979=1026.776,128.547,393.231,168.455,46.701,158.736
C07980=1026.782,128.795,393.211,168.458,46.697,158.736
C07981=1026.788,129.044,393.191,168.460,46.694,158.735
C07982=1026.794,129.294,393.171,168.463,46.691,158.735
C07983=1026.800,129.542,393.151,168.466,46.687,158.734
C07984=1026.806,129.792,393.131,168.469,46.684,158.734
C07985=1026.812,130.040,393.111,168.472,46.680,158.734
C07986=1026.818,130.290,393.090,168.475,46.677,158.734
C07987=1026.824,130.539,393.070,168.477,46.673,158.733
C07988=1026.829,130.788,393.050,168.480,46.670,158.733
C07989=1026.835,131.038,393.029,168.483,46.667,158.733
C07990=1026.841,131.287,393.009,168.486,46.663,158.732
C07991=1026.847,131.536,392.988,168.488,46.660,158.732
C07992=1026.853,131.785,392.968,168.492,46.657,158.731
C07993=1026.858,132.034,392.947,168.494,46.653,158.731
C07994=1026.865,132.282,392.927,168.498,46.650,158.731
C07995=1026.870,132.532,392.906,168.500,46.647,158.730
C07996=1026.877,132.781,392.886,168.502,46.643,158.730
C07997=1026.882,133.030,392.865,168.506,46.640,158.730
C07998=1026.888,133.279,392.845,168.509,46.636,158.730
C07999=1026.894,133.528,392.824,168.511,46.633,158.729
C08000=1026.900,133.777,392.804,168.514,46.630,158.729
C08001=1026.905,134.026,392.783,168.517,46.626,158.728
C08002=1026.912,134.276,392.763,168.520,46.623,158.728
C08003=1026.917,134.524,392.742,168.523,46.619,158.728
C08004=1026.923,134.773,392.721,168.525,46.616,158.727
C08005=1026.929,135.023,392.701,168.528,46.613,158.727
C08006=1026.934,135.272,392.680,168.531,46.609,158.727
C08007=1026.941,135.521,392.659,168.534,46.606,158.727
C08008=1026.947,135.770,392.639,168.537,46.602,158.726
C08009=1026.953,136.019,392.619,168.539,46.599,158.726
C08010=1026.958,136.269,392.598,168.542,46.596,158.726
C08011=1026.964,136.517,392.576,168.545,46.592,158.725
C08012=1026.970,136.766,392.556,168.548,46.589,158.725
C08013=1026.976,137.016,392.536,168.551,46.586,158.725
C08014=1026.982,137.264,392.515,168.553,46.582,158.724
C08015=1026.988,137.514,392.494,168.556,46.579,158.724
C08016=1026.993,137.763,392.473,168.559,46.576,158.724
C08017=1027.000,138.011,392.453,168.562,46.572,158.723
C08018=1027.005,138.261,392.432,168.565,46.569,158.723
C08019=1027.011,138.509,392.411,168.568,46.565,158.723
C08020=1027.018,138.759,392.390,168.571,46.562,158.722
C08021=1027.023,139.008,392.370,168.574,46.559,158.722
C08022=1027.029,139.257,392.348,168.577,46.556,158.722
C08023=1027.034,139.506,392.327,168.580,46.552,158.721
C08024=1027.041,139.790,392.303,168.583,46.548,158.721
C08025=1027.048,140.075,392.279,168.586,46.545,158.721
C08026=1027.054,140.359,392.255,168.590,46.541,158.720
C08027=1027.061,140.643,392.232,168.592,46.537,158.720
C08028=1027.067,140.892,392.211,168.596,46.534,158.720
C08029=1027.072,141.142,392.190,168.599,46.530,158.719
C08030=1027.079,141.390,392.169,168.602,46.527,158.719
C08031=1027.084,141.640,392.148,168.604,46.524,158.719
C08032=1027.090,141.888,392.127,168.607,46.520,158.718
C08033=1027.096,142.137,392.105,168.610,46.517,158.718
C08034=1027.101,142.386,392.085,168.613,46.514,158.718
C08035=1027.108,142.635,392.064,168.616,46.511,158.718
C08036=1027.114,142.884,392.043,168.619,46.507,158.717
C08037=1027.120,143.134,392.022,168.621,46.504,158.717
C08038=1027.125,143.383,392.001,168.624,46.501,158.716
C08039=1027.131,143.632,391.980,168.627,46.498,158.716
C08040=1027.137,143.880,391.959,168.630,46.494,158.716
C08041=1027.143,144.130,391.938,168.634,46.491,158.716
C08042=1027.149,144.379,391.917,168.636,46.487,158.715
C08043=1027.155,144.628,391.895,168.639,46.484,158.715
C08044=1027.160,144.877,391.874,168.642,46.481,158.715
C08045=1027.166,145.126,391.853,168.645,46.477,158.714
C08046=1027.172,145.375,391.833,168.648,46.474,158.714
C08047=1027.179,145.624,391.811,168.651,46.471,158.714
C08048=1027.184,145.873,391.790,168.654,46.468,158.713
C08049=1027.190,146.122,391.769,168.657,46.464,158.713
C08050=1027.196,146.372,391.747,168.660,46.461,158.713
C08051=1027.202,146.620,391.726,168.662,46.458,158.712
C08052=1027.208,146.869,391.704,168.665,46.455,158.712
C08053=1027.213,147.118,391.684,168.668,46.451,158.712
C08054=1027.219,147.368,391.662,168.671,46.448,158.712
C08055=1027.225,147.616,391.641,168.674,46.444,158.711
C08056=1027.231,147.865,391.619,168.678,46.441,158.711
C08057=1027.237,148.114,391.598,168.681,46.438,158.711
C08058=1027.242,148.364,391.577,168.683,46.435,158.710
C08059=1027.249,148.613,391.556,168.686,46.432,158.710
C08060=1027.254,148.861,391.534,168.689,46.428,158.710
C08061=1027.260,149.111,391.513,168.692,46.425,158.710
C08062=1027.266,149.359,391.491,168.695,46.422,158.709
C08063=1027.272,149.608,391.470,168.698,46.419,158.709
C08064=1027.278,149.857,391.449,168.701,46.415,158.709
C08065=1027.284,150.107,391.428,168.704,46.412,158.708
C08066=1027.290,150.356,391.406,168.707,46.409,158.708
C08067=1027.295,150.604,391.385,168.710,46.406,158.708
C08068=1027.301,150.854,391.362,168.713,46.403,158.707
C08069=1027.306,151.102,391.341,168.716,46.399,158.707
C08070=1027.312,151.352,391.320,168.719,46.396,158.707
C08071=1027.319,151.601,391.298,168.722,46.392,158.706
C08072=1027.324,151.849,391.277,168.725,46.389,158.706
C08073=1027.330,152.098,391.255,168.728,46.386,158.706
C08074=1027.336,152.348,391.233,168.731,46.383,158.706
C08075=1027.342,152.596,391.212,168.735,46.380,158.705
C08076=1027.348,152.845,391.190,168.737,46.376,158.705
C08077=1027.354,153.094,391.169,168.740,46.373,158.705
C08078=1027.360,153.343,391.148,168.743,46.370,158.704
C08079=1027.365,153.593,391.125,168.746,46.367,158.704
C08080=1027.371,153.841,391.104,168.749,46.364,158.704
C08081=1027.377,154.090,391.082,168.752,46.360,158.704
C08082=1027.383,154.340,391.061,168.755,46.357,158.703
C08083=1027.388,154.588,391.039,168.759,46.354,158.703
C08084=1027.394,154.838,391.017,168.761,46.350,158.703
C08085=1027.400,155.087,390.996,168.765,46.347,158.703
C08086=1027.406,155.335,390.974,168.768,46.344,158.702
C08087=1027.411,155.585,390.952,168.770,46.341,158.702
C08088=1027.418,155.868,390.927,168.774,46.337,158.702
C08089=1027.425,156.153,390.902,168.777,46.334,158.701
C08090=1027.432,156.437,390.878,168.781,46.330,158.701
C08091=1027.438,156.720,390.852,168.784,46.327,158.701
C08092=1027.444,156.970,390.831,168.787,46.323,158.700
C08093=1027.450,157.218,390.810,168.790,46.320,158.700
C08094=1027.456,157.467,390.787,168.793,46.317,158.700
C08095=1027.462,157.716,390.765,168.796,46.313,158.699
C08096=1027.468,157.965,390.743,168.800,46.310,158.699
C08097=1027.474,158.214,390.722,168.803,46.307,158.699
C08098=1027.480,158.463,390.700,168.806,46.304,158.699
C08099=1027.485,158.712,390.677,168.809,46.301,158.698
C08100=1027.492,158.961,390.656,168.812,46.297,158.698
C08101=1027.497,159.210,390.635,168.815,46.294,158.698
C08102=1027.503,159.459,390.612,168.818,46.291,158.698
C08103=1027.509,159.708,390.590,168.822,46.288,158.697
C08104=1027.515,159.957,390.568,168.825,46.285,158.697
C08105=1027.520,160.206,390.545,168.827,46.282,158.697
C08106=1027.526,160.455,390.524,168.830,46.279,158.696
C08107=1027.531,160.704,390.501,168.833,46.276,158.696
C08108=1027.536,160.953,390.479,168.836,46.273,158.696
C08109=1027.543,161.202,390.457,168.840,46.270,158.696
C08110=1027.548,161.451,390.434,168.843,46.267,158.696
C08111=1027.554,161.700,390.412,168.846,46.264,158.695
C08112=1027.560,161.948,390.390,168.849,46.261,158.695
C08113=1027.565,162.198,390.368,168.852,46.257,158.695
C08114=1027.571,162.446,390.345,168.856,46.255,158.694
C08115=1027.576,162.696,390.323,168.858,46.252,158.694
C08116=1027.582,162.944,390.301,168.861,46.249,158.694
C08117=1027.587,163.193,390.278,168.864,46.246,158.694
C08118=1027.593,163.442,390.255,168.868,46.243,158.694
C08119=1027.600,163.691,390.233,168.871,46.240,158.693
C08120=1027.604,163.940,390.211,168.874,46.236,158.693
C08121=1027.610,164.189,390.188,168.877,46.233,158.693
C08122=1027.616,164.438,390.166,168.880,46.230,158.692
C08123=1027.622,164.687,390.144,168.883,46.227,158.692
C08124=1027.628,164.936,390.121,168.887,46.224,158.692
C08125=1027.633,165.184,390.099,168.890,46.221,158.692
C08126=1027.639,165.433,390.076,168.893,46.219,158.692
C08127=1027.645,165.682,390.054,168.896,46.216,158.691
C08128=1027.650,165.931,390.031,168.899,46.212,158.691
C08129=1027.656,166.180,390.008,168.903,46.209,158.691
C08130=1027.662,166.429,389.987,168.906,46.206,158.691
C08131=1027.668,166.678,389.964,168.909,46.203,158.690
C08132=1027.673,166.927,389.942,168.912,46.200,158.690
C08133=1027.679,167.176,389.920,168.915,46.197,158.690
C08134=1027.685,167.425,389.897,168.919,46.194,158.690
C08135=1027.691,167.674,389.874,168.922,46.191,158.689
C08136=1027.696,167.923,389.851,168.925,46.188,158.689
C08137=1027.703,168.172,389.829,168.928,46.185,158.689
C08138=1027.708,168.421,389.806,168.931,46.182,158.689
C08139=1027.714,168.670,389.784,168.935,46.179,158.688
C08140=1027.720,168.918,389.762,168.938,46.176,158.688
C08141=1027.725,169.167,389.739,168.941,46.173,158.688
C08142=1027.731,169.416,389.716,168.944,46.170,158.688
C08143=1027.736,169.665,389.694,168.947,46.166,158.687
C08144=1027.743,169.914,389.671,168.951,46.163,158.687
C08145=1027.749,170.163,389.648,168.954,46.160,158.687
C08146=1027.754,170.412,389.626,168.957,46.157,158.687
C08147=1027.760,170.661,389.603,168.960,46.154,158.686
C08148=1027.766,170.910,389.581,168.963,46.151,158.686
C08149=1027.772,171.159,389.558,168.967,46.148,158.686
C08150=1027.778,171.408,389.535,168.970,46.146,158.686
C08151=1027.783,171.656,389.512,168.973,46.143,158.685
C08152=1027.790,171.940,389.487,168.977,46.139,158.685
C08153=1027.796,172.223,389.461,168.980,46.135,158.685
C08154=1027.804,172.507,389.435,168.984,46.132,158.685
C08155=1027.811,172.791,389.410,168.988,46.128,158.684
C08156=1027.816,173.039,389.387,168.992,46.125,158.684
C08157=1027.822,173.288,389.364,168.995,46.122,158.684
C08158=1027.828,173.537,389.341,168.998,46.119,158.684
C08159=1027.834,173.786,389.318,169.001,46.116,158.683
C08160=1027.840,174.035,389.296,169.005,46.113,158.683
C08161=1027.846,174.284,389.273,169.008,46.110,158.683
C08162=1027.851,174.533,389.250,169.011,46.107,158.683
C08163=1027.858,174.781,389.227,169.014,46.104,158.682
C08164=1027.864,175.030,389.204,169.018,46.101,158.682
C08165=1027.869,175.280,389.182,169.021,46.098,158.682
C08166=1027.875,175.528,389.159,169.025,46.095,158.682
C08167=1027.880,175.777,389.136,169.028,46.092,158.681
C08168=1027.887,176.026,389.114,169.031,46.089,158.681
C08169=1027.893,176.275,389.091,169.034,46.086,158.681
C08170=1027.899,176.524,389.068,169.038,46.083,158.681
C08171=1027.905,176.773,389.045,169.041,46.080,158.680
C08172=1027.911,177.022,389.022,169.045,46.077,158.680
C08173=1027.917,177.270,388.999,169.048,46.073,158.680
C08174=1027.923,177.519,388.976,169.051,46.070,158.680
C08175=1027.929,177.768,388.953,169.055,46.067,158.679
C08176=1027.935,178.017,388.930,169.058,46.064,158.679
C08177=1027.941,178.265,388.907,169.061,46.061,158.679
C08178=1027.947,178.515,388.884,169.064,46.058,158.679
C08179=1027.953,178.764,388.861,169.069,46.055,158.679
C08180=1027.959,179.013,388.838,169.072,46.052,158.678
C08181=1027.965,179.261,388.816,169.075,46.049,158.678
C08182=1027.971,179.510,388.793,169.078,46.046,158.678
C08183=1027.977,179.759,388.770,169.082,46.043,158.678
C08184=1027.983,180.008,388.746,169.086,46.040,158.678
C08185=1027.990,180.257,388.724,169.089,46.037,158.677
C08186=1027.995,180.506,388.701,169.092,46.034,158.677
C08187=1028.001,180.755,388.678,169.095,46.031,158.677
C08188=1028.007,181.003,388.655,169.098,46.028,158.676
C08189=1028.013,181.253,388.631,169.103,46.025,158.676
C08190=1028.020,181.501,388.608,169.106,46.022,158.676
C08191=1028.026,181.750,388.585,169.109,46.019,158.676
C08192=1028.032,181.999,388.563,169.112,46.016,158.676
C08193=1028.037,182.248,388.540,169.116,46.013,158.675
C08194=1028.044,182.497,388.516,169.120,46.010,158.675
C08195=1028.050,182.745,388.493,169.123,46.007,158.675
C08196=1028.055,182.994,388.470,169.126,46.004,158.675
C08197=1028.061,183.243,388.446,169.130,46.001,158.674
C08198=1028.067,183.493,388.422,169.133,45.999,158.674
C08199=1028.073,183.742,388.399,169.136,45.996,158.674
C08200=1028.079,183.990,388.375,169.140,45.993,158.674
C08201=1028.084,184.239,388.352,169.144,45.990,158.674
C08202=1028.090,184.487,388.328,169.147,45.987,158.674
C08203=1028.095,184.737,388.304,169.151,45.984,158.673
C08204=1028.101,184.986,388.281,169.154,45.981,158.673
C08205=1028.107,185.234,388.257,169.157,45.979,158.673
C08206=1028.112,185.483,388.234,169.161,45.976,158.673
C08207=1028.118,185.731,388.210,169.164,45.973,158.673
C08208=1028.124,185.981,388.186,169.168,45.970,158.673
C08209=1028.130,186.229,388.162,169.171,45.967,158.672
C08210=1028.136,186.478,388.139,169.175,45.965,158.672
C08211=1028.141,186.727,388.115,169.178,45.962,158.672
C08212=1028.148,186.976,388.091,169.181,45.959,158.672
C08213=1028.153,187.225,388.068,169.185,45.957,158.672
C08214=1028.159,187.473,388.044,169.189,45.954,158.672
C08215=1028.165,187.722,388.020,169.192,45.951,158.671
C08216=1028.171,188.006,387.993,169.197,45.948,158.671
C08217=1028.177,188.289,387.966,169.200,45.945,158.671
C08218=1028.184,188.571,387.939,169.204,45.941,158.671
C08219=1028.191,188.855,387.911,169.209,45.938,158.671
C08220=1028.197,189.103,387.888,169.212,45.935,158.670
C08221=1028.202,189.352,387.864,169.215,45.932,158.670
C08222=1028.209,189.601,387.840,169.220,45.930,158.670
C08223=1028.215,189.849,387.817,169.223,45.927,158.670
C08224=1028.220,190.099,387.793,169.226,45.924,158.670
C08225=1028.226,190.348,387.769,169.230,45.922,158.670
C08226=1028.232,190.596,387.745,169.233,45.919,158.669
C08227=1028.238,190.844,387.721,169.237,45.916,158.669
C08228=1028.244,191.094,387.696,169.240,45.913,158.669
C08229=1028.249,191.343,387.673,169.244,45.911,158.669
C08230=1028.255,191.591,387.650,169.247,45.908,158.669
C08231=1028.261,191.840,387.625,169.251,45.904,158.668
C08232=1028.267,192.088,387.602,169.255,45.902,158.668
C08233=1028.273,192.338,387.577,169.258,45.899,158.668
C08234=1028.279,192.586,387.553,169.262,45.896,158.668
C08235=1028.284,192.835,387.530,169.266,45.894,158.668
C08236=1028.291,193.084,387.506,169.269,45.891,158.668
C08237=1028.297,193.332,387.482,169.272,45.888,158.667
C08238=1028.303,193.582,387.457,169.277,45.885,158.667
C08239=1028.309,193.830,387.434,169.280,45.883,158.667
C08240=1028.314,194.079,387.409,169.283,45.880,158.667
C08241=1028.321,194.328,387.385,169.288,45.877,158.667
C08242=1028.326,194.576,387.361,169.291,45.874,158.667
C08243=1028.333,194.825,387.337,169.295,45.872,158.667
C08244=1028.339,195.073,387.314,169.298,45.869,158.666
C08245=1028.345,195.323,387.289,169.302,45.866,158.666
C08246=1028.351,195.571,387.265,169.306,45.864,158.666
C08247=1028.357,195.820,387.241,169.309,45.861,158.666
C08248=1028.363,196.069,387.217,169.313,45.858,158.666
C08249=1028.369,196.318,387.192,169.317,45.855,158.666
C08250=1028.375,196.566,387.169,169.320,45.852,158.665
C08251=1028.381,196.815,387.144,169.324,45.849,158.665
C08252=1028.387,197.064,387.120,169.328,45.847,158.665
C08253=1028.392,197.313,387.096,169.332,45.844,158.665
C08254=1028.399,197.561,387.072,169.336,45.842,158.665
C08255=1028.405,197.810,387.048,169.339,45.839,158.665
C08256=1028.410,198.059,387.024,169.343,45.835,158.664
C08257=1028.417,198.308,387.000,169.347,45.833,158.664
C08258=1028.422,198.556,386.976,169.350,45.830,158.664
C08259=1028.429,198.805,386.951,169.354,45.828,158.664
C08260=1028.435,199.055,386.927,169.358,45.825,158.664
C08261=1028.441,199.303,386.903,169.362,45.822,158.664
C08262=1028.447,199.552,386.878,169.365,45.820,158.664
C08263=1028.453,199.800,386.854,169.369,45.817,158.663
C08264=1028.459,200.049,386.830,169.373,45.814,158.663
C08265=1028.466,200.298,386.806,169.376,45.811,158.663
C08266=1028.471,200.547,386.781,169.380,45.809,158.663
C08267=1028.477,200.795,386.756,169.384,45.806,158.663
C08268=1028.483,201.044,386.732,169.388,45.804,158.663
C08269=1028.488,201.293,386.707,169.391,45.801,158.663
C08270=1028.495,201.541,386.683,169.396,45.798,158.663
C08271=1028.501,201.790,386.658,169.399,45.796,158.662
C08272=1028.507,202.039,386.633,169.403,45.793,158.662
C08273=1028.512,202.287,386.608,169.407,45.790,158.662
C08274=1028.518,202.537,386.584,169.410,45.788,158.662
C08275=1028.524,202.784,386.559,169.415,45.785,158.662
C08276=1028.530,203.034,386.535,169.418,45.783,158.662
C08277=1028.537,203.282,386.510,169.422,45.781,158.662
C08278=1028.542,203.531,386.485,169.426,45.777,158.662
C08279=1028.548,203.780,386.461,169.429,45.775,158.662
C08280=1028.573,204.825,386.356,169.801,45.878,158.724
C08281=1028.583,205.203,386.316,169.805,45.876,158.724
C08282=1028.594,205.582,386.277,169.809,45.873,158.724
C08283=1028.604,205.959,386.238,169.814,45.870,158.724
C08284=1028.614,206.337,386.198,169.818,45.867,158.724
C08285=1028.620,206.585,386.172,169.821,45.866,158.724
C08286=1028.627,206.834,386.145,169.823,45.864,158.723
C08287=1028.634,207.082,386.119,169.826,45.862,158.723
C08288=1028.641,207.331,386.093,169.830,45.860,158.723
C08289=1028.648,207.579,386.067,169.832,45.859,158.723
C08290=1028.654,207.828,386.040,169.835,45.857,158.723
C08291=1028.660,208.076,386.014,169.838,45.855,158.723
C08292=1028.667,208.325,385.988,169.840,45.853,158.723
C08293=1028.674,208.573,385.962,169.844,45.852,158.723
C08294=1028.681,208.822,385.935,169.846,45.850,158.723
C08295=1028.687,209.071,385.909,169.849,45.848,158.723
C08296=1028.694,209.319,385.882,169.852,45.846,158.723
C08297=1028.700,209.567,385.856,169.855,45.845,158.723
C08298=1028.707,209.816,385.830,169.858,45.843,158.723
C08299=1028.713,210.064,385.803,169.861,45.841,158.723
C08300=1028.720,210.313,385.777,169.863,45.839,158.723
C08301=1028.727,210.562,385.750,169.866,45.838,158.723
C08302=1028.733,210.810,385.724,169.869,45.836,158.723
C08303=1028.740,211.059,385.697,169.872,45.834,158.723
C08304=1028.747,211.307,385.671,169.875,45.833,158.723
C08305=1028.753,211.556,385.643,169.877,45.831,158.722
C08306=1028.760,211.804,385.617,169.880,45.830,158.722
C08307=1028.766,212.053,385.590,169.884,45.827,158.722
C08308=1028.773,212.301,385.564,169.887,45.826,158.722
C08309=1028.779,212.550,385.537,169.889,45.825,158.722
C08310=1028.786,212.799,385.511,169.892,45.823,158.722
C08311=1028.793,213.047,385.485,169.896,45.821,158.722
C08312=1028.800,213.295,385.457,169.898,45.820,158.722
C08313=1028.806,213.543,385.431,169.901,45.818,158.722
C08314=1028.812,213.792,385.404,169.904,45.816,158.722
C08315=1028.820,214.041,385.378,169.906,45.815,158.722
C08316=1028.825,214.289,385.351,169.910,45.813,158.722
C08317=1028.833,214.537,385.324,169.913,45.811,158.722
C08318=1028.839,214.786,385.297,169.915,45.810,158.722
C08319=1028.846,215.034,385.271,169.918,45.808,158.722
C08320=1028.853,215.283,385.244,169.922,45.806,158.722
C08321=1028.859,215.531,385.217,169.924,45.805,158.722
C08322=1028.866,215.780,385.191,169.927,45.803,158.722
C08323=1028.872,216.029,385.164,169.930,45.802,158.722
C08324=1028.879,216.277,385.138,169.933,45.800,158.722
C08325=1028.886,216.525,385.110,169.936,45.798,158.722
C08326=1028.893,216.774,385.083,169.939,45.797,158.722
C08327=1028.898,217.022,385.057,169.941,45.795,158.722
C08328=1028.906,217.271,385.030,169.945,45.793,158.722
C08329=1028.912,217.520,385.003,169.948,45.792,158.722
C08330=1028.919,217.768,384.976,169.951,45.790,158.722
C08331=1028.926,218.016,384.950,169.953,45.788,158.722
C08332=1028.933,218.265,384.922,169.957,45.787,158.722
C08333=1028.940,218.514,384.896,169.960,45.785,158.722
C08334=1028.946,218.761,384.869,169.962,45.784,158.722
C08335=1028.953,219.010,384.842,169.966,45.782,158.722
C08336=1028.959,219.259,384.815,169.969,45.780,158.722
C08337=1028.970,219.642,384.773,169.973,45.778,158.722
C08338=1028.979,220.026,384.732,169.978,45.775,158.722
C08339=1028.990,220.408,384.690,169.982,45.774,158.722
C08340=1029.000,220.791,384.648,169.987,45.771,158.722
C08341=1029.006,221.040,384.621,169.990,45.770,158.722
C08342=1029.012,221.288,384.594,169.992,45.768,158.722
C08343=1029.020,221.536,384.567,169.996,45.767,158.722
C08344=1029.026,221.785,384.539,169.999,45.765,158.722
C08345=1029.033,222.033,384.512,170.002,45.763,158.722
C08346=1029.039,222.282,384.485,170.004,45.762,158.722
C08347=1029.046,222.530,384.458,170.008,45.760,158.722
C08348=1029.052,222.779,384.431,170.011,45.759,158.722
C08349=1029.059,223.027,384.403,170.014,45.758,158.722
C08350=1029.065,223.275,384.376,170.016,45.756,158.722
C08351=1029.072,223.524,384.349,170.020,45.755,158.722
C08352=1029.079,223.772,384.322,170.023,45.753,158.722
C08353=1029.085,224.021,384.295,170.025,45.751,158.722
C08354=1029.092,224.270,384.267,170.029,45.750,158.722
C08355=1029.099,224.517,384.240,170.032,45.748,158.722
C08356=1029.105,224.766,384.213,170.035,45.747,158.722
C08357=1029.112,225.015,384.185,170.038,45.745,158.722
C08358=1029.119,225.263,384.158,170.041,45.744,158.722
C08359=1029.126,225.512,384.131,170.044,45.743,158.722
C08360=1029.132,225.760,384.104,170.047,45.741,158.722
C08361=1029.138,226.008,384.076,170.051,45.740,158.722
C08362=1029.145,226.257,384.048,170.053,45.738,158.722
C08363=1029.152,226.505,384.022,170.056,45.737,158.722
C08364=1029.159,226.754,383.994,170.060,45.735,158.722
C08365=1029.166,227.002,383.967,170.062,45.733,158.722
C08366=1029.172,227.251,383.939,170.065,45.732,158.722
C08367=1029.179,227.499,383.912,170.069,45.731,158.722
C08368=1029.186,227.747,383.885,170.072,45.729,158.722
C08369=1029.192,227.996,383.857,170.074,45.728,158.722
C08370=1029.199,228.244,383.830,170.078,45.726,158.722
C08371=1029.206,228.492,383.802,170.081,45.725,158.722
C08372=1029.212,228.741,383.774,170.084,45.724,158.722
C08373=1029.219,228.989,383.746,170.087,45.723,158.722
C08374=1029.226,229.238,383.719,170.091,45.721,158.722
C08375=1029.232,229.485,383.691,170.093,45.720,158.722
C08376=1029.238,229.735,383.664,170.096,45.718,158.722
C08377=1029.245,229.983,383.637,170.100,45.717,158.722
C08378=1029.251,230.231,383.609,170.103,45.716,158.722
C08379=1029.258,230.480,383.581,170.105,45.714,158.723
C08380=1029.265,230.728,383.553,170.109,45.713,158.723
C08381=1029.271,230.977,383.526,170.112,45.711,158.723
C08382=1029.278,231.225,383.498,170.115,45.710,158.723
C08383=1029.284,231.474,383.470,170.119,45.709,158.723
C08384=1029.290,231.722,383.442,170.122,45.708,158.723
C08385=1029.297,231.970,383.414,170.124,45.706,158.723
C08386=1029.304,232.218,383.386,170.127,45.705,158.723
C08387=1029.311,232.466,383.358,170.131,45.703,158.723
C08388=1029.317,232.715,383.331,170.134,45.703,158.723
C08389=1029.324,232.963,383.303,170.137,45.701,158.723
C08390=1029.330,233.212,383.274,170.140,45.700,158.723
C08391=1029.337,233.460,383.247,170.143,45.698,158.723
C08392=1029.343,233.709,383.219,170.146,45.697,158.723
C08393=1029.354,234.084,383.177,170.151,45.695,158.723
C08394=1029.364,234.459,383.135,170.156,45.693,158.723
C08395=1029.373,234.835,383.092,170.160,45.691,158.724
C08396=1029.383,235.211,383.050,170.166,45.689,158.724
C08397=1029.390,235.459,383.022,170.169,45.688,158.724
C08398=1029.397,235.708,382.994,170.172,45.687,158.724
C08399=1029.404,235.955,382.966,170.175,45.685,158.724
C08400=1029.410,236.204,382.938,170.178,45.684,158.724
C08401=1029.416,236.453,382.910,170.181,45.683,158.724
C08402=1029.423,236.701,382.882,170.185,45.681,158.724
C08403=1029.430,236.949,382.854,170.188,45.680,158.724
C08404=1029.437,237.197,382.826,170.191,45.679,158.724
C08405=1029.443,237.446,382.798,170.195,45.678,158.724
C08406=1029.450,237.694,382.769,170.197,45.676,158.724
C08407=1029.456,237.942,382.742,170.200,45.675,158.724
C08408=1029.463,238.191,382.714,170.204,45.674,158.725
C08409=1029.469,238.439,382.685,170.207,45.673,158.725
C08410=1029.476,238.687,382.657,170.211,45.671,158.725
C08411=1029.483,238.936,382.629,170.213,45.670,158.725
C08412=1029.490,239.184,382.601,170.217,45.669,158.725
C08413=1029.496,239.432,382.573,170.220,45.667,158.725
C08414=1029.503,239.680,382.544,170.223,45.666,158.725
C08415=1029.509,239.929,382.516,170.226,45.665,158.725
C08416=1029.517,240.178,382.488,170.230,45.664,158.725
C08417=1029.523,240.426,382.459,170.233,45.663,158.725
C08418=1029.529,240.674,382.432,170.237,45.661,158.725
C08419=1029.536,240.922,382.403,170.239,45.660,158.725
C08420=1029.543,241.170,382.374,170.242,45.659,158.726
C08421=1029.549,241.419,382.346,170.246,45.658,158.726
C08422=1029.556,241.667,382.317,170.249,45.657,158.726
C08423=1029.562,241.916,382.289,170.252,45.656,158.726
C08424=1029.569,242.163,382.261,170.256,45.655,158.726
C08425=1029.575,242.412,382.232,170.259,45.653,158.726
C08426=1029.582,242.660,382.204,170.263,45.652,158.726
C08427=1029.588,242.909,382.174,170.266,45.651,158.726
C08428=1029.595,243.157,382.147,170.269,45.650,158.726
C08429=1029.601,243.405,382.118,170.273,45.649,158.727
C08430=1029.608,243.653,382.089,170.276,45.648,158.727
C08431=1029.614,243.902,382.061,170.278,45.647,158.727
C08432=1029.621,244.150,382.032,170.282,45.646,158.727
C08433=1029.627,244.398,382.003,170.285,45.644,158.727
C08434=1029.635,244.647,381.975,170.289,45.643,158.727
C08435=1029.641,244.895,381.946,170.292,45.642,158.727
C08436=1029.647,245.143,381.917,170.295,45.641,158.727
C08437=1029.653,245.391,381.888,170.299,45.640,158.728
C08438=1029.660,245.639,381.860,170.302,45.639,158.728
C08439=1029.666,245.888,381.831,170.305,45.638,158.728
C08440=1029.673,246.136,381.802,170.309,45.637,158.728
C08441=1029.679,246.384,381.773,170.312,45.636,158.728
C08442=1029.687,246.633,381.744,170.316,45.635,158.728
C08443=1029.693,246.881,381.715,170.318,45.634,158.728
C08444=1029.699,247.129,381.686,170.321,45.633,158.728
C08445=1029.705,247.377,381.657,170.326,45.632,158.729
C08446=1029.712,247.625,381.628,170.328,45.631,158.729
C08447=1029.719,247.874,381.600,170.331,45.630,158.729
C08448=1029.725,248.123,381.571,170.335,45.629,158.729
C08449=1029.734,248.492,381.528,170.340,45.627,158.729
C08450=1029.745,248.861,381.485,170.345,45.626,158.729
C08451=1029.755,249.231,381.442,170.350,45.624,158.730
C08452=1029.764,249.599,381.398,170.355,45.623,158.730
C08453=1029.770,249.848,381.370,170.359,45.622,158.730
C08454=1029.777,250.096,381.340,170.362,45.621,158.730
C08455=1029.784,250.345,381.311,170.365,45.620,158.730
C08456=1029.790,250.593,381.282,170.369,45.619,158.731
C08457=1029.797,250.840,381.253,170.372,45.618,158.731
C08458=1029.804,251.089,381.224,170.376,45.617,158.731
C08459=1029.810,251.337,381.195,170.379,45.616,158.731
C08460=1029.816,251.586,381.166,170.383,45.615,158.731
C08461=1029.824,251.834,381.137,170.386,45.614,158.731
C08462=1029.830,252.082,381.108,170.390,45.613,158.731
C08463=1029.836,252.330,381.079,170.393,45.612,158.732
C08464=1029.843,252.579,381.050,170.396,45.611,158.732
C08465=1029.849,252.827,381.021,170.400,45.610,158.732
C08466=1029.856,253.075,380.992,170.403,45.609,158.732
C08467=1029.864,253.323,380.962,170.407,45.608,158.732
C08468=1029.870,253.571,380.933,170.410,45.608,158.732
C08469=1029.876,253.820,380.904,170.414,45.607,158.733
C08470=1029.883,254.068,380.875,170.416,45.605,158.733
C08471=1029.890,254.316,380.846,170.420,45.604,158.733
C08472=1029.896,254.564,380.816,170.424,45.604,158.733
C08473=1029.903,254.813,380.787,170.428,45.603,158.733
C08474=1029.910,255.061,380.758,170.431,45.602,158.733
C08475=1029.916,255.310,380.728,170.434,45.600,158.733
C08476=1029.923,255.557,380.700,170.437,45.600,158.734
C08477=1029.930,255.805,380.670,170.441,45.599,158.734
C08478=1029.937,256.054,380.641,170.444,45.598,158.734
C08479=1029.943,256.302,380.612,170.449,45.597,158.734
C08480=1029.950,256.550,380.582,170.451,45.596,158.734
C08481=1029.957,256.798,380.553,170.455,45.595,158.735
C08482=1029.964,257.047,380.524,170.458,45.594,158.735
C08483=1029.971,257.294,380.494,170.462,45.593,158.735
C08484=1029.977,257.543,380.465,170.465,45.592,158.735
C08485=1029.984,257.791,380.436,170.470,45.591,158.735
C08486=1029.990,258.039,380.406,170.473,45.591,158.735
C08487=1029.998,258.287,380.377,170.476,45.589,158.736
C08488=1030.004,258.535,380.348,170.479,45.588,158.736
C08489=1030.011,258.784,380.318,170.483,45.587,158.736
C08490=1030.018,259.032,380.289,170.486,45.587,158.736
C08491=1030.025,259.280,380.259,170.490,45.586,158.736
C08492=1030.032,259.528,380.230,170.495,45.585,158.737
C08493=1030.039,259.777,380.201,170.498,45.584,158.737
C08494=1030.046,260.025,380.171,170.502,45.583,158.737
C08495=1030.052,260.273,380.142,170.505,45.582,158.737
C08496=1030.059,260.521,380.112,170.508,45.581,158.737
C08497=1030.065,260.769,380.083,170.511,45.580,158.737
C08498=1030.073,261.017,380.053,170.515,45.579,158.738
C08499=1030.079,261.265,380.024,170.519,45.578,158.738
C08500=1030.086,261.514,379.993,170.523,45.578,158.738
C08501=1030.092,261.761,379.964,170.526,45.577,158.738
C08502=1030.099,262.010,379.934,170.530,45.577,158.739
C08503=1030.106,262.258,379.904,170.534,45.576,158.739
C08504=1030.112,262.506,379.874,170.537,45.575,158.739
C08505=1030.122,262.874,379.829,170.542,45.574,158.739
C08506=1030.132,263.242,379.786,170.548,45.572,158.740
C08507=1030.142,263.610,379.742,170.553,45.572,158.740
C08508=1030.151,263.978,379.697,170.558,45.571,158.740
C08509=1030.159,264.226,379.667,170.563,45.570,158.741
C08510=1030.165,264.474,379.637,170.566,45.569,158.741
C08511=1030.172,264.722,379.607,170.570,45.568,158.741
C08512=1030.178,264.971,379.577,170.573,45.567,158.741
C08513=1030.185,265.219,379.547,170.577,45.567,158.741
C08514=1030.192,265.466,379.517,170.580,45.566,158.742
C08515=1030.199,265.714,379.487,170.584,45.565,158.742
C08516=1030.205,265.963,379.456,170.587,45.565,158.742
C08517=1030.212,266.210,379.427,170.591,45.564,158.742
C08518=1030.219,266.459,379.397,170.595,45.563,158.743
C08519=1030.226,266.707,379.366,170.598,45.563,158.743
C08520=1030.232,266.955,379.336,170.602,45.562,158.743
C08521=1030.239,267.203,379.306,170.606,45.561,158.743
C08522=1030.246,267.450,379.276,170.610,45.561,158.744
C08523=1030.252,267.699,379.245,170.613,45.560,158.744
C08524=1030.259,267.947,379.215,170.617,45.559,158.744
C08525=1030.265,268.195,379.185,170.621,45.559,158.744
C08526=1030.272,268.443,379.155,170.624,45.558,158.745
C08527=1030.279,268.691,379.125,170.628,45.557,158.745
C08528=1030.285,268.939,379.094,170.631,45.556,158.745
C08529=1030.292,269.187,379.064,170.636,45.556,158.745
C08530=1030.299,269.436,379.034,170.640,45.555,158.746
C08531=1030.305,269.684,379.004,170.643,45.554,158.746
C08532=1030.312,269.932,378.974,170.647,45.554,158.746
C08533=1030.319,270.180,378.943,170.650,45.553,158.746
C08534=1030.326,270.428,378.913,170.654,45.553,158.747
C08535=1030.332,270.676,378.882,170.658,45.552,158.747
C08536=1030.339,270.924,378.852,170.661,45.551,158.747
C08537=1030.346,271.172,378.821,170.666,45.551,158.747
C08538=1030.352,271.420,378.791,170.669,45.550,158.748
C08539=1030.359,271.668,378.760,170.673,45.550,158.748
C08540=1030.366,271.916,378.730,170.677,45.549,158.748
C08541=1030.372,272.165,378.699,170.680,45.549,158.749
C08542=1030.378,272.412,378.669,170.684,45.548,158.749
C08543=1030.386,272.660,378.638,170.688,45.548,158.749
C08544=1030.392,272.908,378.607,170.692,45.547,158.749
C08545=1030.399,273.157,378.577,170.696,45.547,158.750
C08546=1030.405,273.404,378.546,170.699,45.546,158.750
C08547=1030.413,273.652,378.516,170.703,45.546,158.750
C08548=1030.419,273.901,378.485,170.707,45.545,158.750
C08549=1030.426,274.149,378.454,170.711,45.545,158.751
C08550=1030.433,274.397,378.423,170.715,45.544,158.751
C08551=1030.439,274.644,378.392,170.718,45.544,158.751
C08552=1030.445,274.892,378.362,170.722,45.543,158.752
C08553=1030.453,275.141,378.332,170.727,45.542,158.752
C08554=1030.459,275.389,378.300,170.730,45.542,158.752
C08555=1030.467,275.637,378.270,170.734,45.541,158.753
C08556=1030.473,275.884,378.239,170.738,45.541,158.753
C08557=1030.479,276.133,378.208,170.741,45.540,158.753
C08558=1030.487,276.380,378.177,170.746,45.540,158.754
C08559=1030.493,276.629,378.147,170.750,45.539,158.754
C08560=1030.500,276.877,378.115,170.753,45.539,158.754
C08561=1030.510,277.249,378.070,170.759,45.538,158.755
C08562=1030.521,277.622,378.023,170.765,45.537,158.755
C08563=1030.530,277.994,377.976,170.771,45.537,158.756
C08564=1030.540,278.367,377.930,170.776,45.536,158.756
C08565=1030.547,278.615,377.898,170.780,45.536,158.756
C08566=1030.554,278.863,377.867,170.785,45.536,158.757
C08567=1030.560,279.111,377.836,170.788,45.535,158.757
C08568=1030.567,279.359,377.805,170.792,45.534,158.757
C08569=1030.573,279.607,377.773,170.796,45.534,158.758
C08570=1030.580,279.855,377.742,170.800,45.534,158.758
C08571=1030.586,280.103,377.711,170.804,45.533,158.758
C08572=1030.593,280.350,377.681,170.808,45.533,158.759
C08573=1030.600,280.598,377.649,170.811,45.533,158.759
C08574=1030.607,280.846,377.618,170.816,45.532,158.759
C08575=1030.614,281.094,377.586,170.820,45.532,158.760
C08576=1030.620,281.342,377.555,170.823,45.531,158.760
C08577=1030.627,281.590,377.524,170.827,45.531,158.760
C08578=1030.633,281.838,377.493,170.832,45.531,158.761
C08579=1030.640,282.086,377.461,170.835,45.531,158.761
C08580=1030.647,282.334,377.430,170.839,45.530,158.761
C08581=1030.654,282.582,377.398,170.844,45.530,158.762
C08582=1030.661,282.830,377.368,170.848,45.530,158.762
C08583=1030.668,283.078,377.336,170.851,45.529,158.762
C08584=1030.675,283.325,377.305,170.855,45.529,158.763
C08585=1030.681,283.573,377.273,170.860,45.528,158.763
C08586=1030.688,283.821,377.242,170.864,45.528,158.764
C08587=1030.695,284.069,377.210,170.867,45.528,158.764
C08588=1030.701,284.317,377.179,170.871,45.528,158.764
C08589=1030.708,284.565,377.148,170.876,45.527,158.765
C08590=1030.715,284.813,377.116,170.880,45.527,158.765
C08591=1030.722,285.061,377.085,170.883,45.527,158.765
C08592=1030.729,285.309,377.053,170.888,45.527,158.766
C08593=1030.736,285.557,377.021,170.892,45.526,158.766
C08594=1030.742,285.805,376.990,170.896,45.526,158.767
C08595=1030.750,286.053,376.959,170.899,45.525,158.767
C08596=1030.756,286.301,376.927,170.904,45.526,158.767
C08597=1030.763,286.548,376.895,170.908,45.525,158.768
C08598=1030.770,286.796,376.864,170.913,45.525,158.768
C08599=1030.776,287.044,376.832,170.916,45.525,158.768
C08600=1030.783,287.292,376.801,170.920,45.525,158.769
C08601=1030.790,287.539,376.769,170.924,45.524,158.769
C08602=1030.797,287.787,376.737,170.929,45.524,158.770
C08603=1030.803,288.036,376.705,170.932,45.524,158.770
C08604=1030.810,288.283,376.673,170.936,45.523,158.770
C08605=1030.817,288.531,376.641,170.941,45.523,158.771
C08606=1030.824,288.779,376.610,170.945,45.523,158.771
C08607=1030.831,289.026,376.578,170.950,45.523,158.772
C08608=1030.838,289.274,376.546,170.953,45.523,158.772
C08609=1030.844,289.523,376.514,170.957,45.523,158.772
C08610=1030.851,289.771,376.482,170.962,45.522,158.773
C08611=1030.858,290.018,376.450,170.966,45.522,158.773
C08612=1030.865,290.266,376.418,170.969,45.522,158.773
C08613=1030.872,290.514,376.387,170.974,45.522,158.774
C08614=1030.878,290.761,376.354,170.978,45.522,158.774
C08615=1030.885,291.010,376.322,170.982,45.522,158.775
C08616=1030.892,291.258,376.291,170.987,45.521,158.775
C08617=1030.903,291.642,376.241,170.993,45.521,158.776
C08618=1030.913,292.027,376.191,171.000,45.521,158.776
C08619=1030.924,292.411,376.141,171.006,45.521,158.777
C08620=1030.935,292.797,376.091,171.012,45.521,158.778
C08621=1030.941,293.044,376.059,171.016,45.521,158.778
C08622=1030.948,293.292,376.026,171.021,45.521,158.779
C08623=1030.955,293.540,375.995,171.025,45.521,158.779
C08624=1030.962,293.788,375.962,171.030,45.521,158.780
C08625=1030.969,294.035,375.930,171.034,45.520,158.780
C08626=1030.975,294.283,375.898,171.037,45.520,158.780
C08627=1030.982,294.531,375.865,171.042,45.521,158.781
C08628=1030.989,294.779,375.833,171.046,45.520,158.781
C08629=1030.996,295.026,375.800,171.051,45.521,158.782
C08630=1031.002,295.274,375.768,171.055,45.520,158.782
C08631=1031.010,295.522,375.735,171.060,45.521,158.783
C08632=1031.016,295.770,375.703,171.063,45.521,158.783
C08633=1031.022,296.018,375.670,171.068,45.521,158.784
C08634=1031.029,296.266,375.638,171.072,45.521,158.784
C08635=1031.036,296.513,375.605,171.076,45.521,158.785
C08636=1031.042,296.761,375.572,171.081,45.521,158.785
C08637=1031.049,297.009,375.539,171.085,45.521,158.786
C08638=1031.056,297.256,375.507,171.089,45.521,158.786
C08639=1031.062,297.504,375.474,171.093,45.521,158.786
C08640=1031.069,297.752,375.441,171.098,45.521,158.787
C08641=1031.076,297.999,375.409,171.102,45.522,158.788
C08642=1031.082,298.247,375.376,171.107,45.521,158.788
C08643=1031.089,298.495,375.343,171.111,45.522,158.789
C08644=1031.097,298.742,375.310,171.116,45.521,158.789
C08645=1031.103,298.990,375.278,171.119,45.522,158.789
C08646=1031.110,299.238,375.244,171.124,45.522,158.790
C08647=1031.116,299.486,375.212,171.128,45.522,158.790
C08648=1031.124,299.733,375.179,171.133,45.522,158.791
C08649=1031.130,299.981,375.146,171.137,45.522,158.791
C08650=1031.136,300.229,375.114,171.142,45.522,158.792
C08651=1031.144,300.476,375.080,171.146,45.522,158.792
C08652=1031.151,300.724,375.048,171.151,45.523,158.793
C08653=1031.158,300.972,375.015,171.155,45.523,158.794
C08654=1031.164,301.220,374.982,171.159,45.523,158.794
C08655=1031.171,301.468,374.949,171.163,45.523,158.794
C08656=1031.178,301.714,374.916,171.168,45.523,158.795
C08657=1031.185,301.963,374.883,171.172,45.524,158.796
C08658=1031.192,302.210,374.851,171.177,45.523,158.796
C08659=1031.199,302.458,374.817,171.181,45.524,158.796
C08660=1031.205,302.705,374.784,171.186,45.524,158.797
C08661=1031.212,302.954,374.751,171.190,45.524,158.798
C08662=1031.220,303.200,374.718,171.195,45.524,158.798
C08663=1031.227,303.449,374.685,171.199,45.524,158.799
C08664=1031.233,303.696,374.652,171.204,45.525,158.799
C08665=1031.241,303.944,374.619,171.208,45.525,158.800
C08666=1031.248,304.192,374.586,171.213,45.525,158.800
C08667=1031.254,304.439,374.552,171.218,45.525,158.801
C08668=1031.261,304.687,374.519,171.222,45.525,158.801
C08669=1031.268,304.934,374.487,171.226,45.525,158.802
C08670=1031.275,305.182,374.453,171.231,45.526,158.802
C08671=1031.282,305.430,374.420,171.236,45.526,158.803
C08672=1031.289,305.677,374.387,171.240,45.526,158.803
C08673=1031.301,306.079,374.333,171.247,45.527,158.804
C08674=1031.312,306.481,374.279,171.255,45.527,158.805
C08675=1031.324,306.883,374.225,171.262,45.527,158.806
C08676=1031.335,307.285,374.171,171.270,45.527,158.807
C08677=1031.342,307.532,374.139,171.274,45.528,158.807
C08678=1031.349,307.780,374.105,171.279,45.528,158.808
C08679=1031.356,308.027,374.071,171.283,45.528,158.808
C08680=1031.363,308.276,374.038,171.288,45.529,158.809
C08681=1031.371,308.522,374.005,171.293,45.529,158.810
C08682=1031.378,308.770,373.971,171.297,45.529,158.810
C08683=1031.385,309.018,373.938,171.302,45.530,158.811
C08684=1031.392,309.266,373.904,171.306,45.530,158.811
C08685=1031.399,309.513,373.871,171.311,45.530,158.812
C08686=1031.407,309.760,373.838,171.316,45.531,158.813
C08687=1031.413,310.009,373.804,171.320,45.531,158.813
C08688=1031.421,310.256,373.771,171.326,45.531,158.814
C08689=1031.429,310.504,373.737,171.330,45.532,158.814
C08690=1031.435,310.751,373.704,171.335,45.532,158.815
C08691=1031.442,310.998,373.670,171.340,45.532,158.815
C08692=1031.450,311.246,373.636,171.344,45.532,158.816
C08693=1031.457,311.494,373.602,171.349,45.533,158.816
C08694=1031.464,311.741,373.569,171.354,45.534,158.817
C08695=1031.470,311.989,373.535,171.358,45.534,158.818
C08696=1031.477,312.236,373.501,171.363,45.534,158.818
C08697=1031.484,312.484,373.467,171.368,45.535,158.819
C08698=1031.491,312.732,373.433,171.372,45.535,158.820
C08699=1031.497,312.979,373.399,171.377,45.536,158.820
C08700=1031.504,313.226,373.364,171.382,45.537,158.821
C08701=1031.511,313.474,373.330,171.386,45.537,158.821
C08702=1031.518,313.722,373.296,171.391,45.538,158.822
C08703=1031.525,313.970,373.262,171.396,45.538,158.823
C08704=1031.532,314.217,373.228,171.401,45.539,158.824
C08705=1031.539,314.464,373.194,171.406,45.539,158.824
C08706=1031.545,314.712,373.159,171.411,45.540,158.825
C08707=1031.553,314.959,373.126,171.415,45.540,158.825
C08708=1031.559,315.207,373.090,171.420,45.541,158.826
C08709=1031.567,315.454,373.057,171.425,45.541,158.827
C08710=1031.574,315.702,373.023,171.430,45.542,158.827
C08711=1031.581,315.949,372.988,171.434,45.543,158.828
C08712=1031.588,316.197,372.954,171.439,45.543,158.829
C08713=1031.595,316.445,372.920,171.444,45.544,158.829
C08714=1031.602,316.692,372.885,171.450,45.544,158.830
C08715=1031.609,316.940,372.851,171.454,45.545,158.831
C08716=1031.616,317.187,372.816,171.459,45.546,158.831
C08717=1031.623,317.435,372.782,171.464,45.546,158.832
C08718=1031.630,317.682,372.748,171.468,45.547,158.833
C08719=1031.637,317.930,372.713,171.473,45.548,158.833
C08720=1031.644,318.177,372.679,171.478,45.548,158.834
C08721=1031.651,318.425,372.644,171.484,45.549,158.835
C08722=1031.658,318.672,372.610,171.489,45.549,158.835
C08723=1031.666,318.920,372.576,171.493,45.550,158.836
C08724=1031.672,319.167,372.541,171.498,45.551,158.837
C08725=1031.680,319.415,372.507,171.503,45.552,158.837
C08726=1031.686,319.662,372.472,171.507,45.552,158.838
C08727=1031.694,319.909,372.437,171.513,45.552,158.839
C08728=1031.700,320.157,372.403,171.518,45.553,158.839
C08729=1031.713,320.564,372.346,171.526,45.554,158.840
C08730=1031.724,320.971,372.289,171.535,45.556,158.842
C08731=1031.736,321.377,372.232,171.543,45.556,158.843
C08732=1031.748,321.784,372.175,171.551,45.558,158.844
C08733=1031.755,322.032,372.141,171.556,45.559,158.845
C08734=1031.762,322.279,372.106,171.561,45.560,158.845
C08735=1031.770,322.527,372.071,171.566,45.560,158.846
C08736=1031.778,322.774,372.036,171.570,45.561,158.847
C08737=1031.784,323.021,372.001,171.576,45.561,158.847
C08738=1031.792,323.268,371.967,171.581,45.562,158.848
C08739=1031.798,323.516,371.932,171.586,45.563,158.849
C08740=1031.806,323.764,371.897,171.592,45.564,158.850
C08741=1031.813,324.011,371.862,171.597,45.565,158.850
C08742=1031.821,324.258,371.828,171.601,45.565,158.851
C08743=1031.828,324.506,371.792,171.606,45.566,158.852
C08744=1031.836,324.753,371.758,171.612,45.566,158.853
C08745=1031.843,325.000,371.723,171.617,45.567,158.853
C08746=1031.850,325.249,371.688,171.622,45.568,158.854
C08747=1031.858,325.496,371.653,171.627,45.569,158.855
C08748=1031.865,325.743,371.618,171.632,45.570,158.855
C08749=1031.873,325.991,371.583,171.637,45.571,158.856
C08750=1031.880,326.238,371.548,171.643,45.571,158.857
C08751=1031.887,326.485,371.513,171.648,45.572,158.858
C08752=1031.894,326.733,371.478,171.653,45.573,158.858
C08753=1031.902,326.980,371.443,171.659,45.574,158.859
C08754=1031.909,327.228,371.408,171.663,45.575,158.860
C08755=1031.917,327.475,371.373,171.668,45.575,158.861
C08756=1031.925,327.723,371.337,171.674,45.576,158.861
C08757=1031.932,327.970,371.303,171.679,45.577,158.862
C08758=1031.939,328.217,371.267,171.684,45.578,158.863
C08759=1031.946,328.465,371.232,171.690,45.579,158.864
C08760=1031.953,328.712,371.196,171.695,45.580,158.865
C08761=1031.961,328.960,371.161,171.700,45.581,158.865
C08762=1031.968,329.207,371.125,171.706,45.582,158.866
C08763=1031.976,329.455,371.090,171.711,45.583,158.867
C08764=1031.983,329.702,371.055,171.716,45.584,158.868
C08765=1031.990,329.949,371.019,171.722,45.585,158.869
C08766=1031.997,330.197,370.983,171.727,45.586,158.869
C08767=1032.004,330.444,370.947,171.731,45.587,158.870
C08768=1032.011,330.692,370.912,171.738,45.588,158.871
C08769=1032.019,330.938,370.876,171.742,45.589,158.872
C08770=1032.027,331.185,370.841,171.747,45.590,158.873
C08771=1032.034,331.433,370.805,171.753,45.591,158.874
C08772=1032.041,331.680,370.769,171.758,45.592,158.874
C08773=1032.049,331.928,370.734,171.764,45.593,158.875
C08774=1032.056,332.175,370.698,171.769,45.594,158.876
C08775=1032.064,332.423,370.662,171.774,45.596,158.877
C08776=1032.070,332.670,370.626,171.780,45.596,158.878
C08777=1032.078,332.917,370.590,171.785,45.598,158.879
C08778=1032.085,333.164,370.554,171.791,45.598,158.879
C08779=1032.092,333.412,370.519,171.796,45.600,158.880
C08780=1032.100,333.660,370.483,171.802,45.600,158.881
C08781=1032.108,333.906,370.447,171.807,45.602,158.882
C08782=1032.116,334.153,370.411,171.812,45.603,158.883
C08783=1032.123,334.402,370.376,171.818,45.604,158.884
C08784=1032.130,334.648,370.340,171.823,45.605,158.884
C08785=1032.142,335.050,370.280,171.833,45.607,158.886
C08786=1032.153,335.453,370.222,171.842,45.609,158.887
C08787=1032.165,335.855,370.163,171.850,45.611,158.889
C08788=1032.178,336.257,370.104,171.859,45.613,158.890
C08789=1032.185,336.504,370.068,171.865,45.614,158.891
C08790=1032.193,336.752,370.032,171.870,45.615,158.892
C08791=1032.200,336.999,369.996,171.876,45.616,158.893
C08792=1032.207,337.246,369.959,171.881,45.618,158.894
C08793=1032.215,337.494,369.923,171.888,45.619,158.895
C08794=1032.222,337.741,369.886,171.893,45.621,158.896
C08795=1032.230,337.987,369.850,171.899,45.622,158.897
C08796=1032.237,338.235,369.814,171.904,45.623,158.897
C08797=1032.245,338.482,369.777,171.910,45.624,158.898
C08798=1032.252,338.730,369.741,171.915,45.625,158.899
C08799=1032.260,338.977,369.704,171.921,45.627,158.900
C08800=1032.267,339.224,369.668,171.926,45.628,158.901
C08801=1032.275,339.471,369.632,171.932,45.629,158.902
C08802=1032.282,339.718,369.595,171.937,45.631,158.903
C08803=1032.289,339.966,369.559,171.944,45.632,158.904
C08804=1032.297,340.213,369.522,171.950,45.633,158.905
C08805=1032.305,340.460,369.485,171.955,45.635,158.906
C08806=1032.313,340.707,369.449,171.961,45.636,158.907
C08807=1032.320,340.955,369.412,171.966,45.637,158.908
C08808=1032.328,341.203,369.375,171.972,45.639,158.908
C08809=1032.335,341.449,369.339,171.977,45.640,158.909
C08810=1032.342,341.696,369.302,171.984,45.641,158.910
C08811=1032.350,341.943,369.265,171.990,45.643,158.911
C08812=1032.357,342.190,369.228,171.995,45.645,158.912
C08813=1032.365,342.438,369.191,172.001,45.646,158.913
C08814=1032.373,342.685,369.155,172.006,45.647,158.914
C08815=1032.380,342.932,369.118,172.013,45.648,158.915
C08816=1032.388,343.179,369.081,172.019,45.650,158.916
C08817=1032.395,343.426,369.043,172.024,45.652,158.917
C08818=1032.403,343.674,369.007,172.030,45.653,158.918
C08819=1032.410,343.921,368.969,172.036,45.655,158.919
C08820=1032.418,344.168,368.933,172.042,45.656,158.920
C08821=1032.426,344.415,368.896,172.048,45.657,158.921
C08822=1032.433,344.662,368.859,172.053,45.660,158.922
C08823=1032.441,344.909,368.822,172.059,45.661,158.923
C08824=1032.448,345.156,368.784,172.066,45.662,158.924
C08825=1032.455,345.403,368.747,172.071,45.664,158.925
C08826=1032.463,345.650,368.710,172.077,45.665,158.926
C08827=1032.471,345.898,368.672,172.084,45.667,158.927
C08828=1032.479,346.145,368.635,172.089,45.668,158.928
C08829=1032.486,346.392,368.598,172.095,45.670,158.929
C08830=1032.494,346.639,368.561,172.101,45.671,158.930
C08831=1032.502,346.886,368.523,172.107,45.674,158.931
C08832=1032.510,347.133,368.486,172.113,45.675,158.932
C08833=1032.517,347.380,368.449,172.119,45.677,158.934
C08834=1032.525,347.627,368.411,172.125,45.678,158.934
C08835=1032.533,347.875,368.374,172.131,45.680,158.936
C08836=1032.541,348.121,368.337,172.137,45.681,158.937
C08837=1032.548,348.369,368.299,172.143,45.683,158.938
C08838=1032.556,348.616,368.262,172.149,45.685,158.939
C08839=1032.564,348.863,368.225,172.155,45.686,158.940
C08840=1032.571,349.110,368.186,172.161,45.688,158.941
C08841=1032.584,349.509,368.125,172.172,45.691,158.943
C08842=1032.596,349.907,368.065,172.181,45.693,158.944
C08843=1032.608,350.307,368.004,172.191,45.696,158.946
C08844=1032.621,350.706,367.943,172.201,45.699,158.948
C08845=1032.628,350.953,367.905,172.207,45.701,158.949
C08846=1032.636,351.199,367.868,172.213,45.703,158.950
C08847=1032.644,351.447,367.830,172.219,45.705,158.951
C08848=1032.652,351.693,367.792,172.226,45.707,158.952
C08849=1032.659,351.941,367.754,172.232,45.708,158.953
C08850=1032.667,352.188,367.715,172.238,45.709,158.954
C08851=1032.675,352.435,367.678,172.244,45.712,158.956
C08852=1032.683,352.681,367.640,172.250,45.713,158.957
C08853=1032.691,352.929,367.602,172.257,45.715,158.958
C08854=1032.698,353.175,367.564,172.263,45.717,158.959
C08855=1032.706,353.423,367.525,172.269,45.719,158.960
C08856=1032.714,353.669,367.489,172.276,45.720,158.961
C08857=1032.722,353.917,367.450,172.282,45.723,158.963
C08858=1032.730,354.163,367.412,172.288,45.725,158.964
C08859=1032.738,354.410,367.373,172.294,45.727,158.965
C08860=1032.745,354.658,367.336,172.301,45.728,158.966
C08861=1032.754,354.904,367.298,172.307,45.730,158.967
C08862=1032.762,355.151,367.259,172.314,45.732,158.968
C08863=1032.770,355.398,367.221,172.320,45.734,158.969
C08864=1032.778,355.645,367.182,172.327,45.736,158.971
C08865=1032.785,355.893,367.145,172.333,45.738,158.972
C08866=1032.793,356.139,367.106,172.340,45.740,158.973
C08867=1032.801,356.386,367.068,172.345,45.742,158.974
C08868=1032.809,356.633,367.029,172.352,45.744,158.975
C08869=1032.817,356.880,366.991,172.358,45.746,158.976
C08870=1032.824,357.127,366.953,172.365,45.748,158.978
C08871=1032.833,357.373,366.913,172.371,45.750,158.979
C08872=1032.841,357.620,366.875,172.378,45.752,158.980
C08873=1032.849,357.867,366.836,172.384,45.754,158.981
C08874=1032.857,358.114,366.798,172.391,45.756,158.983
C08875=1032.865,358.361,366.759,172.398,45.758,158.984
C08876=1032.872,358.608,366.721,172.404,45.760,158.985
C08877=1032.881,358.855,366.682,172.411,45.763,158.986
C08878=1032.889,359.102,366.643,172.417,45.764,158.987
C08879=1032.897,359.348,366.605,172.424,45.767,158.989
C08880=1032.905,359.595,366.566,172.430,45.769,158.990
C08881=1032.913,359.842,366.527,172.437,45.771,158.991
C08882=1032.921,360.089,366.488,172.443,45.773,158.992
C08883=1032.928,360.336,366.449,172.450,45.775,158.994
C08884=1032.937,360.583,366.410,172.457,45.777,158.995
C08885=1032.945,360.830,366.371,172.463,45.779,158.996
C08886=1032.953,361.076,366.332,172.470,45.782,158.998
C08887=1032.961,361.323,366.294,172.478,45.784,158.999
C08888=1032.969,361.569,366.255,172.484,45.786,159.000
C08889=1032.977,361.817,366.215,172.491,45.788,159.002
C08890=1032.985,362.064,366.176,172.498,45.790,159.003
C08891=1032.993,362.311,366.137,172.504,45.792,159.004
C08892=1033.000,362.557,366.098,172.511,45.795,159.005
C08893=1033.009,362.804,366.059,172.518,45.797,159.007
C08894=1033.017,363.050,366.019,172.524,45.800,159.008
C08895=1033.025,363.298,365.980,172.531,45.802,159.009
C08896=1033.033,363.544,365.941,172.538,45.804,159.011
C08897=1033.046,363.950,365.876,172.550,45.808,159.013
C08898=1033.060,364.355,365.812,172.561,45.812,159.015
C08899=1033.073,364.759,365.746,172.572,45.816,159.017
C08900=1033.087,365.164,365.682,172.583,45.820,159.019
C08901=1033.094,365.411,365.642,172.590,45.822,159.021
C08902=1033.103,365.658,365.603,172.597,45.824,159.022
C08903=1033.111,365.905,365.563,172.604,45.827,159.023
C08904=1033.119,366.151,365.523,172.611,45.829,159.025
C08905=1033.127,366.398,365.484,172.618,45.832,159.026
C08906=1033.136,366.645,365.445,172.625,45.834,159.028
C08907=1033.144,366.892,365.405,172.632,45.836,159.029
C08908=1033.152,367.138,365.366,172.639,45.839,159.030
C08909=1033.160,367.385,365.326,172.646,45.842,159.032
C08910=1033.168,367.631,365.286,172.653,45.844,159.033
C08911=1033.177,367.878,365.246,172.661,45.846,159.035
C08912=1033.185,368.125,365.206,172.668,45.849,159.036
C08913=1033.194,368.372,365.167,172.674,45.851,159.037
C08914=1033.202,368.618,365.127,172.681,45.854,159.039
C08915=1033.210,368.865,365.087,172.689,45.856,159.040
C08916=1033.219,369.111,365.047,172.696,45.859,159.042
C08917=1033.227,369.358,365.006,172.703,45.861,159.043
C08918=1033.236,369.605,364.967,172.711,45.864,159.044
C08919=1033.243,369.852,364.927,172.718,45.866,159.046
C08920=1033.252,370.098,364.887,172.725,45.869,159.047
C08921=1033.260,370.344,364.846,172.732,45.871,159.049
C08922=1033.269,370.592,364.806,172.739,45.874,159.050
C08923=1033.277,370.838,364.766,172.746,45.877,159.052
C08924=1033.285,371.085,364.726,172.754,45.879,159.053
C08925=1033.293,371.331,364.686,172.761,45.882,159.055
C08926=1033.302,371.577,364.645,172.768,45.885,159.056
C08927=1033.310,371.824,364.605,172.776,45.888,159.058
C08928=1033.318,372.071,364.565,172.783,45.891,159.059
C08929=1033.326,372.317,364.524,172.790,45.893,159.061
C08930=1033.336,372.564,364.484,172.798,45.896,159.062
C08931=1033.344,372.810,364.443,172.805,45.899,159.064
C08932=1033.352,373.057,364.402,172.813,45.901,159.065
C08933=1033.361,373.303,364.362,172.820,45.904,159.067
C08934=1033.369,373.550,364.322,172.828,45.907,159.068
C08935=1033.377,373.797,364.281,172.835,45.910,159.070
C08936=1033.385,374.043,364.240,172.842,45.913,159.071
C08937=1033.395,374.290,364.200,172.850,45.915,159.073
C08938=1033.403,374.536,364.159,172.857,45.918,159.074
C08939=1033.411,374.782,364.119,172.865,45.921,159.076
C08940=1033.420,375.028,364.078,172.872,45.924,159.078
C08941=1033.428,375.275,364.037,172.880,45.926,159.079
C08942=1033.437,375.522,363.996,172.887,45.930,159.081
C08943=1033.446,375.769,363.955,172.895,45.932,159.082
C08944=1033.454,376.015,363.915,172.902,45.935,159.084
C08945=1033.463,376.262,363.874,172.911,45.938,159.085
C08946=1033.471,376.507,363.832,172.919,45.941,159.087
C08947=1033.480,376.754,363.791,172.926,45.944,159.089
C08948=1033.489,377.000,363.751,172.934,45.947,159.090
C08949=1033.497,377.247,363.710,172.941,45.950,159.092
C08950=1033.506,377.494,363.669,172.949,45.953,159.094
C08951=1033.514,377.740,363.628,172.957,45.955,159.095
C08952=1033.524,377.986,363.587,172.964,45.958,159.097
C08953=1033.531,378.199,363.551,172.971,45.961,159.098
C08954=1033.539,378.412,363.516,172.978,45.963,159.100
C08955=1033.545,378.625,363.480,172.985,45.966,159.101
C08956=1033.553,378.838,363.444,172.991,45.970,159.103
C08957=1033.561,379.051,363.408,172.998,45.972,159.104
C08958=1033.568,379.264,363.372,173.005,45.975,159.105
C08959=1033.575,379.477,363.337,173.012,45.977,159.107
C08960=1033.583,379.690,363.301,173.019,45.980,159.108
C08961=1033.591,379.937,363.259,173.027,45.983,159.110
C08962=1033.600,380.182,363.218,173.034,45.986,159.111
C08963=1033.609,380.429,363.176,173.042,45.989,159.113
C08964=1033.618,380.675,363.135,173.051,45.992,159.115
C08965=1033.627,380.921,363.093,173.058,45.996,159.117
C08966=1033.635,381.168,363.052,173.066,45.999,159.118
C08967=1033.644,381.414,363.011,173.075,46.002,159.120
C08968=1033.653,381.660,362.969,173.083,46.005,159.122
C08969=1033.661,381.907,362.927,173.090,46.008,159.123
C08970=1033.670,382.153,362.885,173.098,46.011,159.125
C08971=1033.679,382.400,362.843,173.107,46.015,159.127
C08972=1033.688,382.646,362.801,173.115,46.018,159.129
C08973=1033.696,382.893,362.760,173.122,46.021,159.130
C08974=1033.706,383.138,362.717,173.131,46.024,159.132
C08975=1033.715,383.385,362.675,173.139,46.028,159.134
C08976=1033.724,383.631,362.634,173.147,46.031,159.136
C08977=1033.732,383.877,362.592,173.156,46.034,159.138
C08978=1033.741,384.124,362.550,173.163,46.038,159.139
C08979=1033.751,384.369,362.508,173.171,46.041,159.141
C08980=1033.760,384.616,362.466,173.180,46.044,159.143
C08981=1033.769,384.862,362.424,173.188,46.047,159.145
C08982=1033.777,385.108,362.381,173.197,46.051,159.147
C08983=1033.786,385.355,362.340,173.205,46.054,159.148
C08984=1033.795,385.601,362.298,173.213,46.057,159.150
C08985=1033.804,385.847,362.256,173.222,46.061,159.152
C08986=1033.813,386.093,362.214,173.230,46.064,159.154
C08987=1033.822,386.339,362.171,173.239,46.068,159.156
C08988=1033.832,386.586,362.129,173.247,46.071,159.158
C08989=1033.841,386.832,362.087,173.256,46.074,159.159
C08990=1033.850,387.077,362.044,173.264,46.078,159.161
C08991=1033.859,387.324,362.002,173.272,46.082,159.163
C08992=1033.868,387.571,361.959,173.280,46.085,159.165
C08993=1033.878,387.816,361.917,173.289,46.089,159.167
C08994=1033.886,388.062,361.874,173.297,46.092,159.169
C08995=1033.895,388.309,361.832,173.306,46.096,159.171
C08996=1033.904,388.554,361.790,173.314,46.100,159.173
C08997=1033.913,388.801,361.746,173.324,46.103,159.175
C08998=1033.923,389.047,361.704,173.332,46.106,159.176
C08999=1033.931,389.293,361.661,173.341,46.110,159.178
C09000=1033.941,389.539,361.618,173.350,46.114,159.180
C09001=1033.950,389.785,361.576,173.358,46.117,159.182
C09002=1033.959,390.031,361.533,173.367,46.121,159.184
C09003=1033.969,390.278,361.490,173.376,46.125,159.186
C09004=1033.977,390.524,361.447,173.384,46.129,159.188
C09005=1033.987,390.770,361.403,173.393,46.132,159.190
C09006=1033.996,391.016,361.360,173.402,46.136,159.192
C09007=1034.005,391.261,361.318,173.410,46.140,159.194
C09008=1034.014,391.508,361.274,173.420,46.143,159.196
C09009=1034.024,391.753,361.231,173.429,46.147,159.198
C09010=1034.033,392.000,361.188,173.437,46.151,159.200
C09011=1034.042,392.246,361.145,173.446,46.155,159.202
C09012=1034.051,392.492,361.101,173.455,46.159,159.204
C09013=1034.060,392.726,361.060,173.463,46.162,159.206
C09014=1034.069,392.960,361.019,173.472,46.166,159.208
C09015=1034.078,393.195,360.978,173.481,46.170,159.210
C09016=1034.087,393.430,360.937,173.489,46.173,159.212
C09017=1034.096,393.664,360.895,173.498,46.177,159.214
C09018=1034.105,393.898,360.854,173.507,46.181,159.216
C09019=1034.114,394.134,360.812,173.515,46.184,159.218
C09020=1034.123,394.368,360.771,173.524,46.188,159.220
C09021=1034.132,394.614,360.727,173.533,46.192,159.222
C09022=1034.141,394.860,360.683,173.542,46.196,159.224
C09023=1034.151,395.105,360.640,173.551,46.200,159.226
C09024=1034.160,395.352,360.596,173.560,46.204,159.228
C09025=1034.170,395.598,360.552,173.570,46.208,159.230
C09026=1034.179,395.843,360.509,173.579,46.212,159.232
C09027=1034.188,396.089,360.465,173.588,46.216,159.234
C09028=1034.198,396.335,360.421,173.598,46.220,159.237
C09029=1034.207,396.582,360.377,173.607,46.224,159.239
C09030=1034.217,396.827,360.333,173.617,46.228,159.241
C09031=1034.227,397.072,360.289,173.626,46.233,159.243
C09032=1034.236,397.318,360.245,173.635,46.237,159.245
C09033=1034.245,397.565,360.201,173.645,46.241,159.247
C09034=1034.256,397.810,360.157,173.654,46.245,159.250
C09035=1034.265,398.056,360.113,173.664,46.249,159.252
C09036=1034.275,398.302,360.068,173.673,46.253,159.254
C09037=1034.284,398.548,360.024,173.683,46.257,159.256
C09038=1034.294,398.794,359.981,173.692,46.261,159.258
C09039=1034.304,399.039,359.936,173.701,46.265,159.260
C09040=1034.313,399.286,359.892,173.712,46.270,159.263
C09041=1034.323,399.532,359.848,173.721,46.274,159.265
C09042=1034.332,399.777,359.803,173.731,46.278,159.267
C09043=1034.343,400.022,359.759,173.740,46.283,159.270
C09044=1034.352,400.269,359.714,173.750,46.287,159.272
C09045=1034.362,400.514,359.670,173.759,46.292,159.274
C09046=1034.371,400.760,359.625,173.769,46.296,159.276
C09047=1034.381,401.006,359.581,173.779,46.300,159.279
C09048=1034.391,401.251,359.536,173.788,46.304,159.281
C09049=1034.401,401.497,359.491,173.799,46.309,159.283
C09050=1034.410,401.742,359.446,173.809,46.313,159.286
C09051=1034.420,401.989,359.402,173.818,46.317,159.288
C09052=1034.430,402.235,359.357,173.828,46.322,159.290
C09053=1034.440,402.480,359.312,173.838,46.326,159.293
C09054=1034.449,402.726,359.267,173.848,46.331,159.295
C09055=1034.460,402.972,359.222,173.858,46.336,159.297
C09056=1034.470,403.217,359.177,173.868,46.340,159.300
C09057=1034.478,403.463,359.132,173.879,46.345,159.302
C09058=1034.489,403.708,359.086,173.888,46.349,159.305
C09059=1034.499,403.954,359.041,173.898,46.354,159.307
C09060=1034.509,404.200,358.996,173.908,46.358,159.309
C09061=1034.518,404.445,358.951,173.919,46.363,159.312
C09062=1034.529,404.691,358.906,173.929,46.367,159.314
C09063=1034.538,404.937,358.860,173.939,46.372,159.317
C09064=1034.548,405.183,358.815,173.949,46.377,159.319
C09065=1034.558,405.428,358.769,173.959,46.382,159.322
C09066=1034.569,405.674,358.724,173.970,46.386,159.324
C09067=1034.579,405.919,358.679,173.980,46.390,159.326
C09068=1034.588,406.166,358.633,173.990,46.396,159.329
C09069=1034.598,406.403,358.588,174.001,46.400,159.331
C09070=1034.608,406.640,358.545,174.010,46.405,159.334
C09071=1034.618,406.877,358.501,174.020,46.409,159.336
C09072=1034.627,407.114,358.457,174.031,46.414,159.339
C09073=1034.637,407.355,358.412,174.041,46.419,159.341
C09074=1034.647,407.596,358.367,174.052,46.423,159.344
C09075=1034.658,407.837,358.322,174.062,46.427,159.346
C09076=1034.667,408.077,358.278,174.071,46.433,159.349
C09077=1034.677,408.318,358.233,174.082,46.437,159.351
C09078=1034.688,408.558,358.187,174.092,46.442,159.354
C09079=1034.698,408.799,358.143,174.103,46.447,159.356
C09080=1034.707,409.040,358.097,174.113,46.452,159.359
C09081=1034.718,409.286,358.051,174.124,46.457,159.361
C09082=1034.728,409.531,358.006,174.135,46.461,159.364
C09083=1034.739,409.776,357.960,174.146,46.466,159.367
C09084=1034.749,410.022,357.914,174.157,46.471,159.369
C09085=1034.760,410.267,357.867,174.167,46.476,159.372
C09086=1034.770,410.513,357.821,174.178,46.481,159.374
C09087=1034.781,410.758,357.775,174.190,46.486,159.377
C09088=1034.791,411.004,357.729,174.201,46.491,159.380
C09089=1034.802,411.249,357.682,174.211,46.496,159.382
C09090=1034.812,411.495,357.636,174.222,46.501,159.385
C09091=1034.822,411.740,357.589,174.234,46.507,159.388
C09092=1034.833,411.986,357.543,174.244,46.512,159.391
C09093=1034.843,412.231,357.496,174.255,46.517,159.393
C09094=1034.854,412.477,357.450,174.267,46.522,159.396
C09095=1034.864,412.722,357.403,174.278,46.527,159.399
C09096=1034.874,412.967,357.355,174.289,46.533,159.402
C09097=1034.885,413.213,357.309,174.300,46.537,159.404
C09098=1034.895,413.458,357.262,174.311,46.543,159.407
C09099=1034.906,413.703,357.216,174.323,46.548,159.410
C09100=1034.917,413.949,357.168,174.334,46.554,159.413
C09101=1034.928,414.194,357.121,174.346,46.558,159.416
